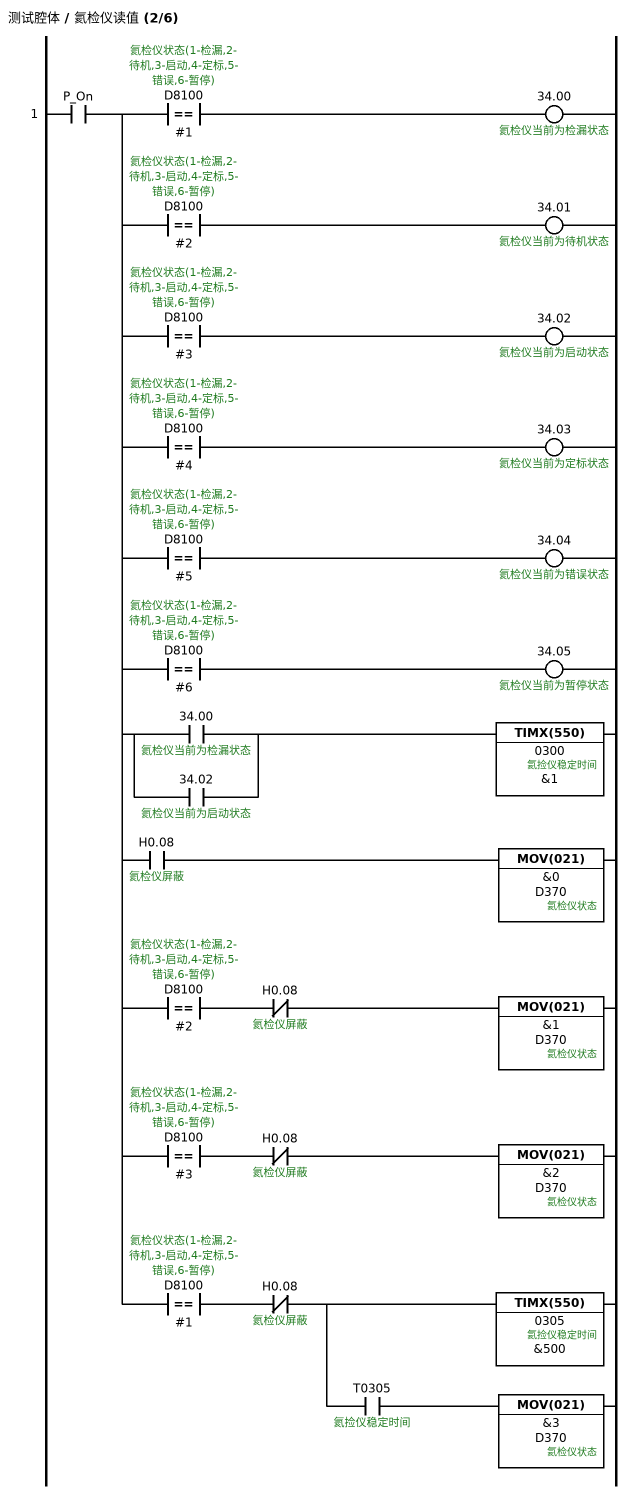
; [picture p144: 测试腔体 / 氦检仪读值, rungs 1-1]
; rung 1
LD P_On
OUT TR0
AND=(300) D8100 #1  ; 氦检仪状态(1-检漏,2-待机,3-启动,4-定标,5-错误,6-暂停)
OUT 34.00  ; 氦检仪当前为检漏状态
LD TR0
AND=(300) D8100 #2  ; 氦检仪状态(1-检漏,2-待机,3-启动,4-定标,5-错误,6-暂停)
OUT 34.01  ; 氦检仪当前为待机状态
LD TR0
AND=(300) D8100 #3  ; 氦检仪状态(1-检漏,2-待机,3-启动,4-定标,5-错误,6-暂停)
OUT 34.02  ; 氦检仪当前为启动状态
LD TR0
AND=(300) D8100 #4  ; 氦检仪状态(1-检漏,2-待机,3-启动,4-定标,5-错误,6-暂停)
OUT 34.03  ; 氦检仪当前为定标状态
LD TR0
AND=(300) D8100 #5  ; 氦检仪状态(1-检漏,2-待机,3-启动,4-定标,5-错误,6-暂停)
OUT 34.04  ; 氦检仪当前为错误状态
LD TR0
AND=(300) D8100 #6  ; 氦检仪状态(1-检漏,2-待机,3-启动,4-定标,5-错误,6-暂停)
OUT 34.05  ; 氦检仪当前为暂停状态
LD TR0
LD 34.00  ; 氦检仪当前为检漏状态
OR 34.02  ; 氦检仪当前为启动状态
ANDLD
TIMX(550) 0300 &1  ; 氦捡仪稳定时间
LD TR0
AND H0.08  ; 氦检仪屏蔽
MOV(021) &0 D370  ; 氦检仪状态
LD TR0
AND=(300) D8100 #2  ; 氦检仪状态(1-检漏,2-待机,3-启动,4-定标,5-错误,6-暂停)
ANDNOT H0.08  ; 氦检仪屏蔽
MOV(021) &1 D370  ; 氦检仪状态
LD TR0
AND=(300) D8100 #3  ; 氦检仪状态(1-检漏,2-待机,3-启动,4-定标,5-错误,6-暂停)
ANDNOT H0.08  ; 氦检仪屏蔽
MOV(021) &2 D370  ; 氦检仪状态
LD TR0
AND=(300) D8100 #1  ; 氦检仪状态(1-检漏,2-待机,3-启动,4-定标,5-错误,6-暂停)
ANDNOT H0.08  ; 氦检仪屏蔽
TIMX(550) 0305 &500  ; 氦捡仪稳定时间
AND T0305  ; 氦捡仪稳定时间
MOV(021) &3 D370  ; 氦检仪状态

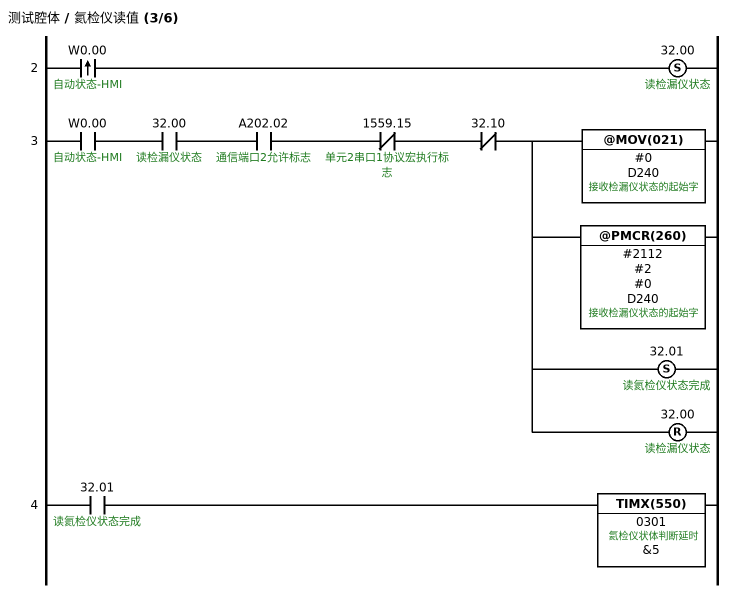
; rung 2
@LD W0.00  ; 自动状态-HMI
SET 32.00  ; 读检漏仪状态
; rung 3
LD W0.00  ; 自动状态-HMI
AND 32.00  ; 读检漏仪状态
AND A202.02  ; 通信端口2允许标志
ANDNOT 1559.15  ; 单元2串口1协议宏执行标志
ANDNOT 32.10
@MOV(021) #0 D240  ; 接收检漏仪状态的起始字
@PMCR(260) #2112 #2 #0 D240  ; 接收检漏仪状态的起始字
SET 32.01  ; 读氦检仪状态完成
RSET 32.00  ; 读检漏仪状态
; rung 4
LD 32.01  ; 读氦检仪状态完成
TIMX(550) 0301 &5  ; 氦检仪状体判断延时

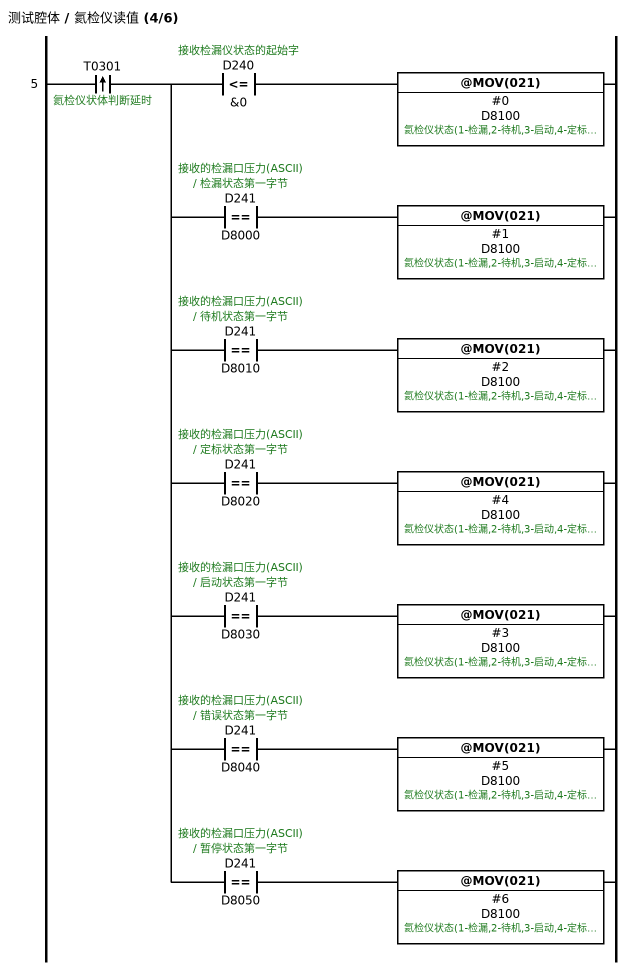
; rung 5
@LD T0301  ; 氦检仪状体判断延时
OUT TR0
AND<=(315) D240 &0  ; 接收检漏仪状态的起始字
@MOV(021) #0 D8100  ; 氦检仪状态(1-检漏,2-待机,3-启动,4-定标,5-错误,6-暂停)
LD TR0
AND=L(301) D241 D8000  ; 接收的检漏口压力(ASCII), 检漏状态第一字节
@MOV(021) #1 D8100  ; 氦检仪状态(1-检漏,2-待机,3-启动,4-定标,5-错误,6-暂停)
LD TR0
AND=L(301) D241 D8010  ; 接收的检漏口压力(ASCII), 待机状态第一字节
@MOV(021) #2 D8100  ; 氦检仪状态(1-检漏,2-待机,3-启动,4-定标,5-错误,6-暂停)
LD TR0
AND=L(301) D241 D8020  ; 接收的检漏口压力(ASCII), 定标状态第一字节
@MOV(021) #4 D8100  ; 氦检仪状态(1-检漏,2-待机,3-启动,4-定标,5-错误,6-暂停)
LD TR0
AND=L(301) D241 D8030  ; 接收的检漏口压力(ASCII), 启动状态第一字节
@MOV(021) #3 D8100  ; 氦检仪状态(1-检漏,2-待机,3-启动,4-定标,5-错误,6-暂停)
LD TR0
AND=L(301) D241 D8040  ; 接收的检漏口压力(ASCII), 错误状态第一字节
@MOV(021) #5 D8100  ; 氦检仪状态(1-检漏,2-待机,3-启动,4-定标,5-错误,6-暂停)
LD TR0
AND=L(301) D241 D8050  ; 接收的检漏口压力(ASCII), 暂停状态第一字节
@MOV(021) #6 D8100  ; 氦检仪状态(1-检漏,2-待机,3-启动,4-定标,5-错误,6-暂停)

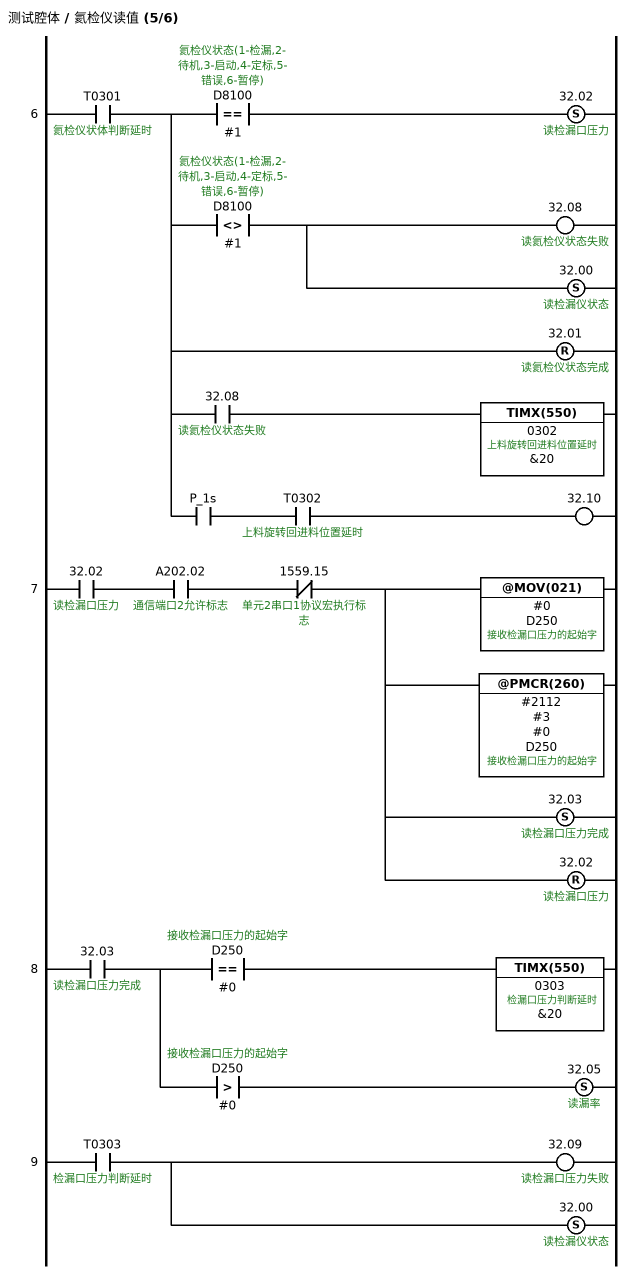
; rung 6
LD T0301  ; 氦检仪状体判断延时
OUT TR0
AND=(300) D8100 #1  ; 氦检仪状态(1-检漏,2-待机,3-启动,4-定标,5-错误,6-暂停)
SET 32.02  ; 读检漏口压力
LD TR0
AND<>(305) D8100 #1  ; 氦检仪状态(1-检漏,2-待机,3-启动,4-定标,5-错误,6-暂停)
OUT 32.08  ; 读氦检仪状态失败
SET 32.00  ; 读检漏仪状态
LD TR0
RSET 32.01  ; 读氦检仪状态完成
AND 32.08  ; 读氦检仪状态失败
TIMX(550) 0302 &20  ; 上料旋转回进料位置延时
LD TR0
AND P_1s
AND T0302  ; 上料旋转回进料位置延时
OUT 32.10
; rung 7
LD 32.02  ; 读检漏口压力
AND A202.02  ; 通信端口2允许标志
ANDNOT 1559.15  ; 单元2串口1协议宏执行标志
@MOV(021) #0 D250  ; 接收检漏口压力的起始字
@PMCR(260) #2112 #3 #0 D250  ; 接收检漏口压力的起始字
SET 32.03  ; 读检漏口压力完成
RSET 32.02  ; 读检漏口压力
; rung 8
LD 32.03  ; 读检漏口压力完成
OUT TR0
AND=(300) D250 #0  ; 接收检漏口压力的起始字
TIMX(550) 0303 &20  ; 检漏口压力判断延时
LD TR0
AND>(320) D250 #0  ; 接收检漏口压力的起始字
SET 32.05  ; 读漏率
; rung 9
LD T0303  ; 检漏口压力判断延时
OUT 32.09  ; 读检漏口压力失败
SET 32.00  ; 读检漏仪状态

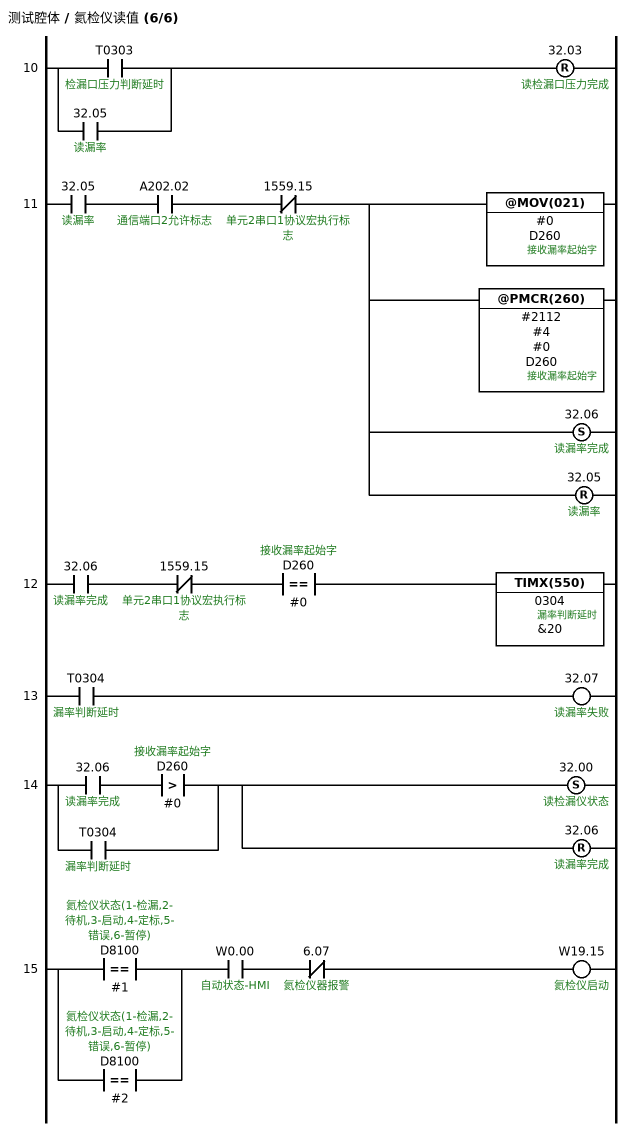
; rung 10
LD T0303  ; 检漏口压力判断延时
OR 32.05  ; 读漏率
RSET 32.03  ; 读检漏口压力完成
; rung 11
LD 32.05  ; 读漏率
AND A202.02  ; 通信端口2允许标志
ANDNOT 1559.15  ; 单元2串口1协议宏执行标志
@MOV(021) #0 D260  ; 接收漏率起始字
@PMCR(260) #2112 #4 #0 D260  ; 接收漏率起始字
SET 32.06  ; 读漏率完成
RSET 32.05  ; 读漏率
; rung 12
LD 32.06  ; 读漏率完成
ANDNOT 1559.15  ; 单元2串口1协议宏执行标志
AND=(300) D260 #0  ; 接收漏率起始字
TIMX(550) 0304 &20  ; 漏率判断延时
; rung 13
LD T0304  ; 漏率判断延时
OUT 32.07  ; 读漏率失败
; rung 14
LD 32.06  ; 读漏率完成
AND>(320) D260 #0  ; 接收漏率起始字
OR T0304  ; 漏率判断延时
SET 32.00  ; 读检漏仪状态
RSET 32.06  ; 读漏率完成
; rung 15
LD=(300) D8100 #1  ; 氦检仪状态(1-检漏,2-待机,3-启动,4-定标,5-错误,6-暂停)
OR=(300) D8100 #2  ; 氦检仪状态(1-检漏,2-待机,3-启动,4-定标,5-错误,6-暂停)
AND W0.00  ; 自动状态-HMI
ANDNOT 6.07  ; 氦检仪器报警
OUT W19.15  ; 氦检仪启动

### Section 外部输出_腔体状态

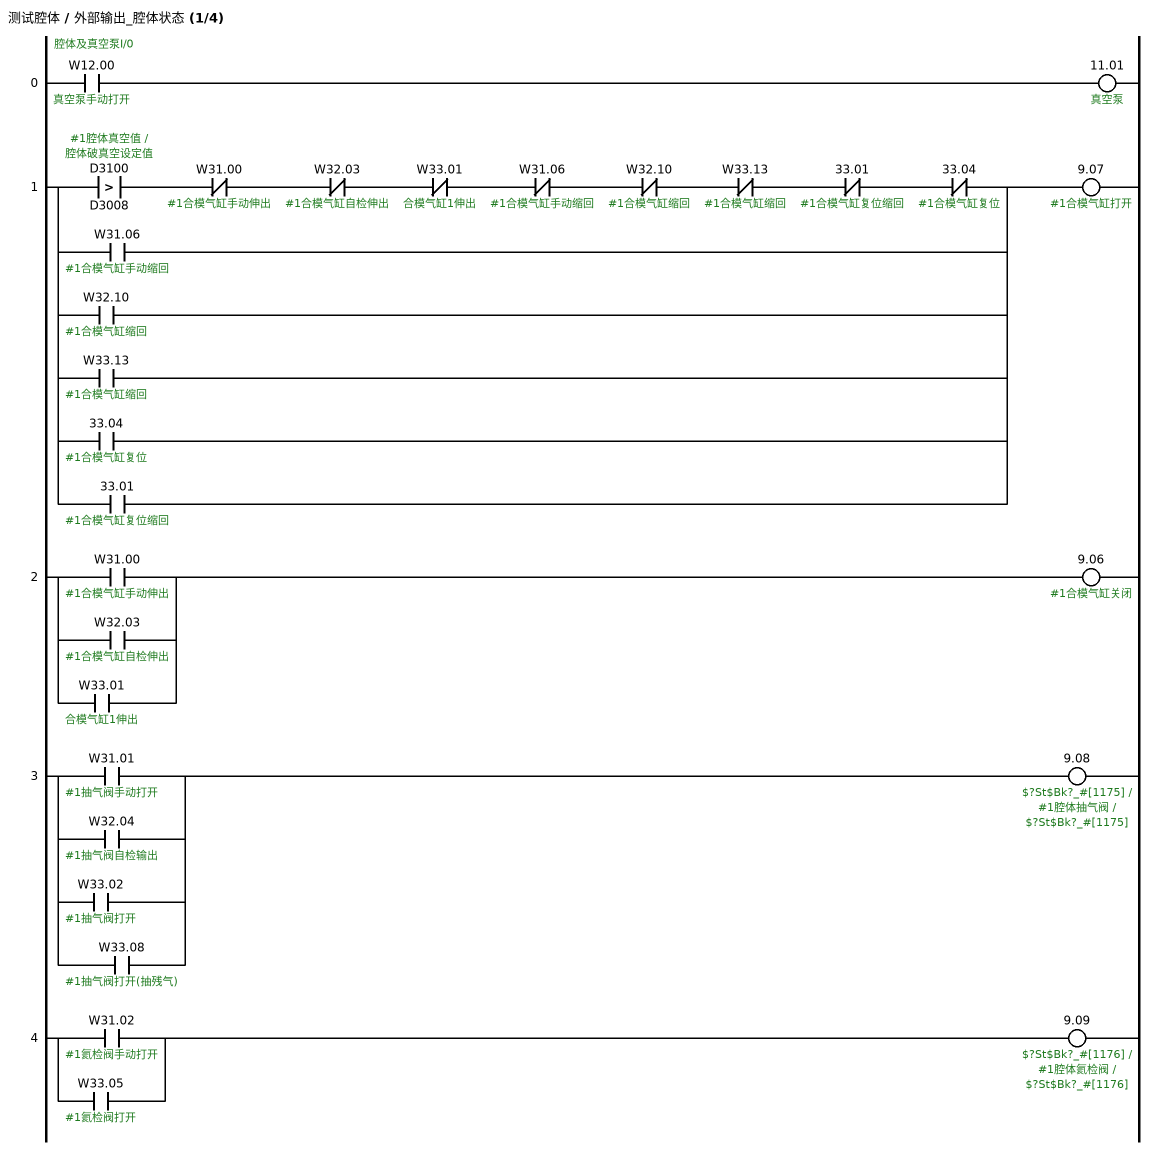
; rung 0: 腔体及真空泵I/0
LD W12.00  ; 真空泵手动打开
OUT 11.01  ; 真空泵
; rung 1
LD>F(333) D3100 D3008  ; #1腔体真空值, 腔体破真空设定值
ANDNOT W31.00  ; #1合模气缸手动伸出
ANDNOT W32.03  ; #1合模气缸自检伸出
ANDNOT W33.01  ; 合模气缸1伸出
ANDNOT W31.06  ; #1合模气缸手动缩回
ANDNOT W32.10  ; #1合模气缸缩回
ANDNOT W33.13  ; #1合模气缸缩回
ANDNOT 33.01  ; #1合模气缸复位缩回
ANDNOT 33.04  ; #1合模气缸复位
OR W31.06  ; #1合模气缸手动缩回
OR W32.10  ; #1合模气缸缩回
OR W33.13  ; #1合模气缸缩回
OR 33.04  ; #1合模气缸复位
OR 33.01  ; #1合模气缸复位缩回
OUT 9.07  ; #1合模气缸打开
; rung 2
LD W31.00  ; #1合模气缸手动伸出
OR W32.03  ; #1合模气缸自检伸出
OR W33.01  ; 合模气缸1伸出
OUT 9.06  ; #1合模气缸关闭
; rung 3
LD W31.01  ; #1抽气阀手动打开
OR W32.04  ; #1抽气阀自检输出
OR W33.02  ; #1抽气阀打开
OR W33.08  ; #1抽气阀打开(抽残气)
OUT 9.08  ; $?St$Bk?_#[1175] / #1腔体抽气阀 / $?St$Bk?_#[1175]
; rung 4
LD W31.02  ; #1氦检阀手动打开
OR W33.05  ; #1氦检阀打开
OUT 9.09  ; $?St$Bk?_#[1176] / #1腔体氦检阀 / $?St$Bk?_#[1176]

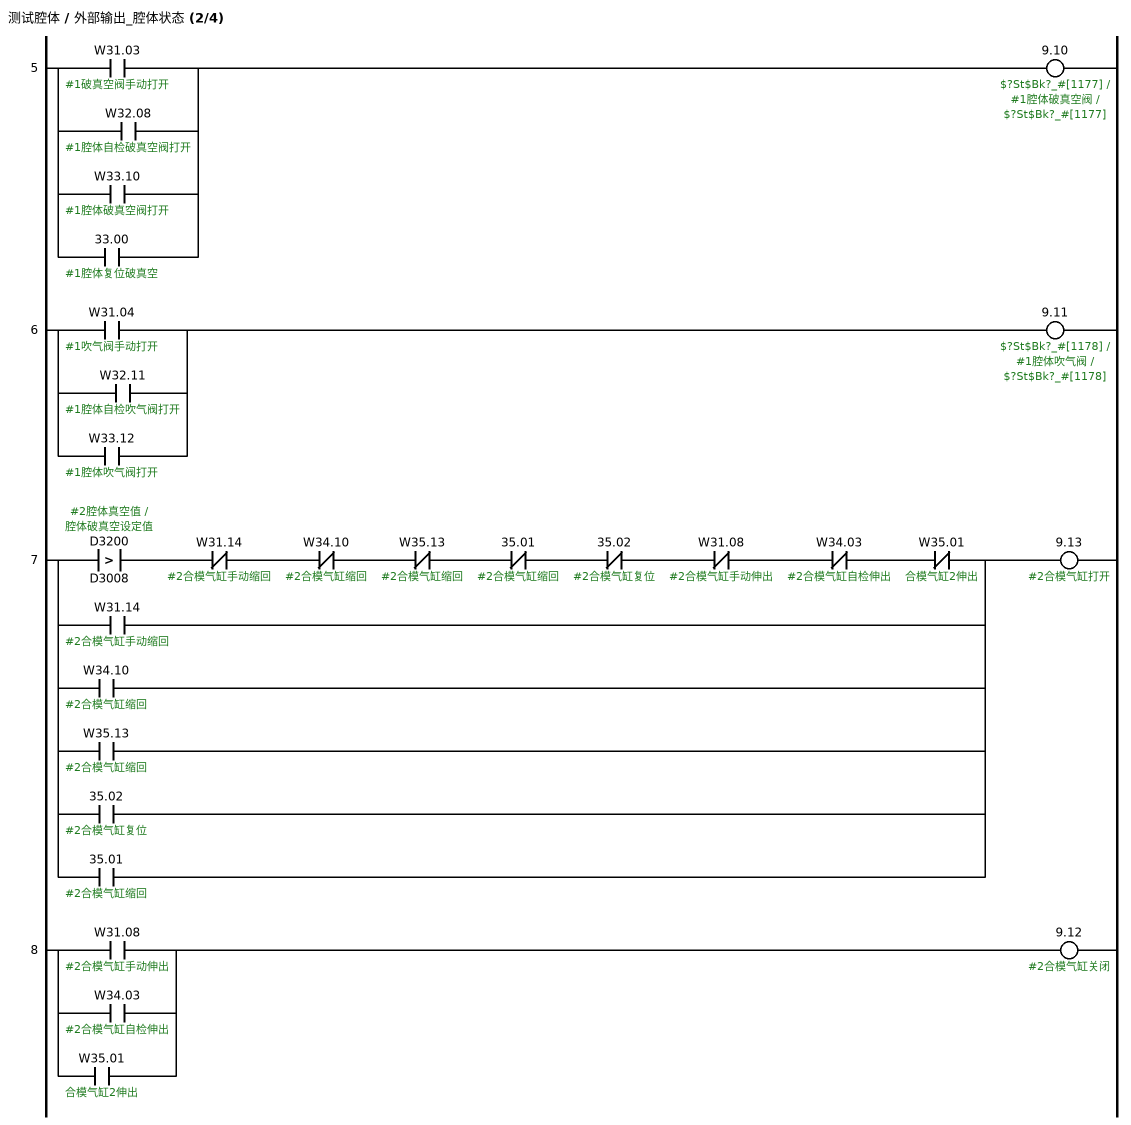
; rung 5
LD W31.03  ; #1破真空阀手动打开
OR W32.08  ; #1腔体自检破真空阀打开
OR W33.10  ; #1腔体破真空阀打开
OR 33.00  ; #1腔体复位破真空
OUT 9.10  ; $?St$Bk?_#[1177] / #1腔体破真空阀 / $?St$Bk?_#[1177]
; rung 6
LD W31.04  ; #1吹气阀手动打开
OR W32.11  ; #1腔体自检吹气阀打开
OR W33.12  ; #1腔体吹气阀打开
OUT 9.11  ; $?St$Bk?_#[1178] / #1腔体吹气阀 / $?St$Bk?_#[1178]
; rung 7
LD>F(333) D3200 D3008  ; #2腔体真空值, 腔体破真空设定值
ANDNOT W31.14  ; #2合模气缸手动缩回
ANDNOT W34.10  ; #2合模气缸缩回
ANDNOT W35.13  ; #2合模气缸缩回
ANDNOT 35.01  ; #2合模气缸缩回
ANDNOT 35.02  ; #2合模气缸复位
ANDNOT W31.08  ; #2合模气缸手动伸出
ANDNOT W34.03  ; #2合模气缸自检伸出
ANDNOT W35.01  ; 合模气缸2伸出
OR W31.14  ; #2合模气缸手动缩回
OR W34.10  ; #2合模气缸缩回
OR W35.13  ; #2合模气缸缩回
OR 35.02  ; #2合模气缸复位
OR 35.01  ; #2合模气缸缩回
OUT 9.13  ; #2合模气缸打开
; rung 8
LD W31.08  ; #2合模气缸手动伸出
OR W34.03  ; #2合模气缸自检伸出
OR W35.01  ; 合模气缸2伸出
OUT 9.12  ; #2合模气缸关闭

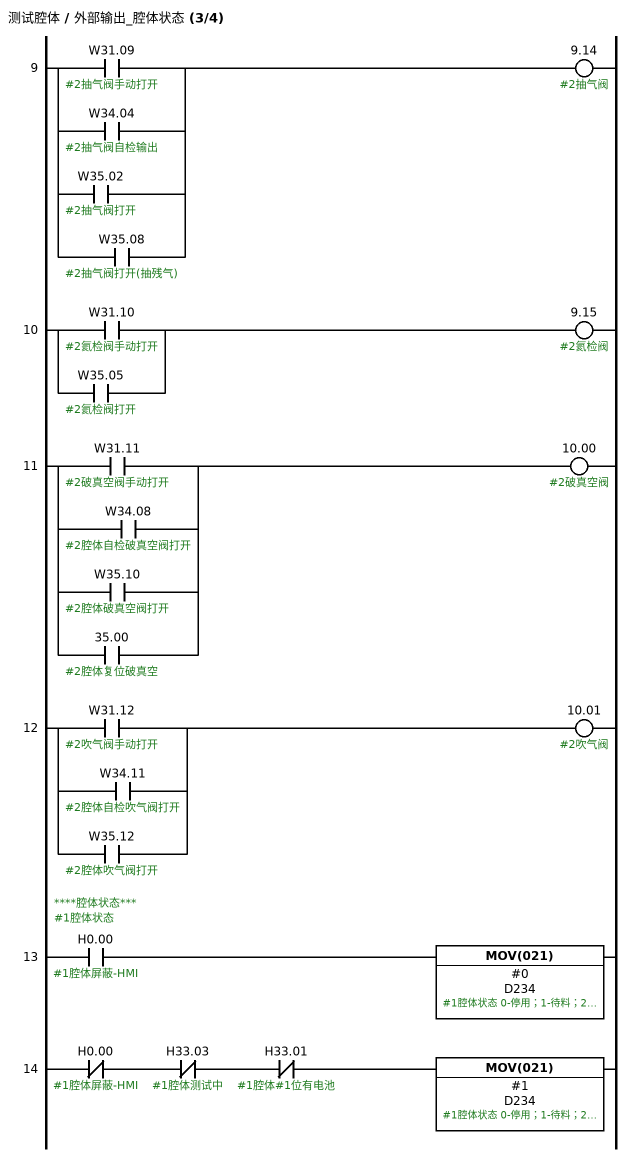
; rung 9
LD W31.09  ; #2抽气阀手动打开
OR W34.04  ; #2抽气阀自检输出
OR W35.02  ; #2抽气阀打开
OR W35.08  ; #2抽气阀打开(抽残气)
OUT 9.14  ; #2抽气阀
; rung 10
LD W31.10  ; #2氦检阀手动打开
OR W35.05  ; #2氦检阀打开
OUT 9.15  ; #2氦检阀
; rung 11
LD W31.11  ; #2破真空阀手动打开
OR W34.08  ; #2腔体自检破真空阀打开
OR W35.10  ; #2腔体破真空阀打开
OR 35.00  ; #2腔体复位破真空
OUT 10.00  ; #2破真空阀
; rung 12
LD W31.12  ; #2吹气阀手动打开
OR W34.11  ; #2腔体自检吹气阀打开
OR W35.12  ; #2腔体吹气阀打开
OUT 10.01  ; #2吹气阀
; rung 13: ****腔体状态*** / #1腔体状态
LD H0.00  ; #1腔体屏蔽-HMI
MOV(021) #0 D234  ; #1腔体状态 0-停用；1-待料；2-测试中；3-测试完成
; rung 14
LDNOT H0.00  ; #1腔体屏蔽-HMI
ANDNOT H33.03  ; #1腔体测试中
ANDNOT H33.01  ; #1腔体#1位有电池
MOV(021) #1 D234  ; #1腔体状态 0-停用；1-待料；2-测试中；3-测试完成

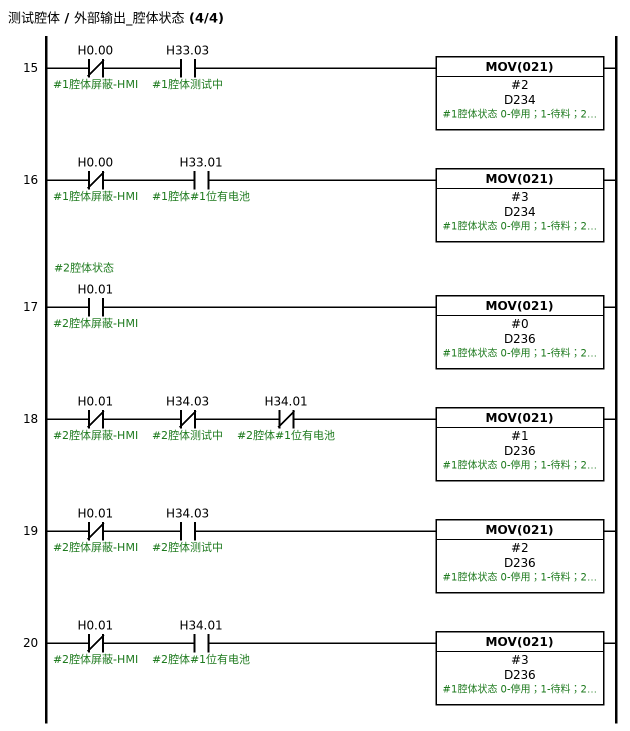
; rung 15
LDNOT H0.00  ; #1腔体屏蔽-HMI
AND H33.03  ; #1腔体测试中
MOV(021) #2 D234  ; #1腔体状态 0-停用；1-待料；2-测试中；3-测试完成
; rung 16
LDNOT H0.00  ; #1腔体屏蔽-HMI
AND H33.01  ; #1腔体#1位有电池
MOV(021) #3 D234  ; #1腔体状态 0-停用；1-待料；2-测试中；3-测试完成
; rung 17: #2腔体状态
LD H0.01  ; #2腔体屏蔽-HMI
MOV(021) #0 D236  ; #1腔体状态 0-停用；1-待料；2-测试中；3-测试完成
; rung 18
LDNOT H0.01  ; #2腔体屏蔽-HMI
ANDNOT H34.03  ; #2腔体测试中
ANDNOT H34.01  ; #2腔体#1位有电池
MOV(021) #1 D236  ; #1腔体状态 0-停用；1-待料；2-测试中；3-测试完成
; rung 19
LDNOT H0.01  ; #2腔体屏蔽-HMI
AND H34.03  ; #2腔体测试中
MOV(021) #2 D236  ; #1腔体状态 0-停用；1-待料；2-测试中；3-测试完成
; rung 20
LDNOT H0.01  ; #2腔体屏蔽-HMI
AND H34.01  ; #2腔体#1位有电池
MOV(021) #3 D236  ; #1腔体状态 0-停用；1-待料；2-测试中；3-测试完成

### Section 报警_复位

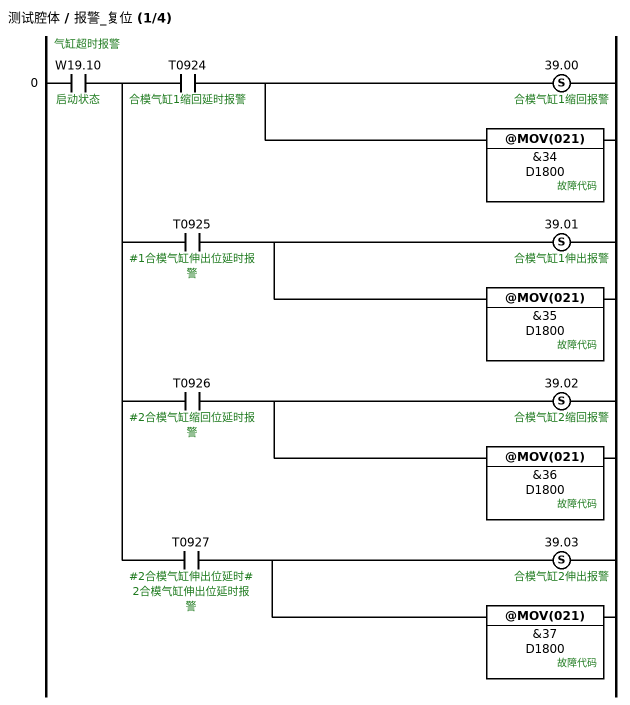
; rung 0: 气缸超时报警
LD W19.10  ; 启动状态
OUT TR0
AND T0924  ; 合模气缸1缩回延时报警
SET 39.00  ; 合模气缸1缩回报警
@MOV(021) &34 D1800  ; 故障代码
LD TR0
AND T0925  ; #1合模气缸伸出位延时报警
SET 39.01  ; 合模气缸1伸出报警
@MOV(021) &35 D1800  ; 故障代码
LD TR0
AND T0926  ; #2合模气缸缩回位延时报警
SET 39.02  ; 合模气缸2缩回报警
@MOV(021) &36 D1800  ; 故障代码
LD TR0
AND T0927  ; #2合模气缸伸出位延时#2合模气缸伸出位延时报警
SET 39.03  ; 合模气缸2伸出报警
@MOV(021) &37 D1800  ; 故障代码

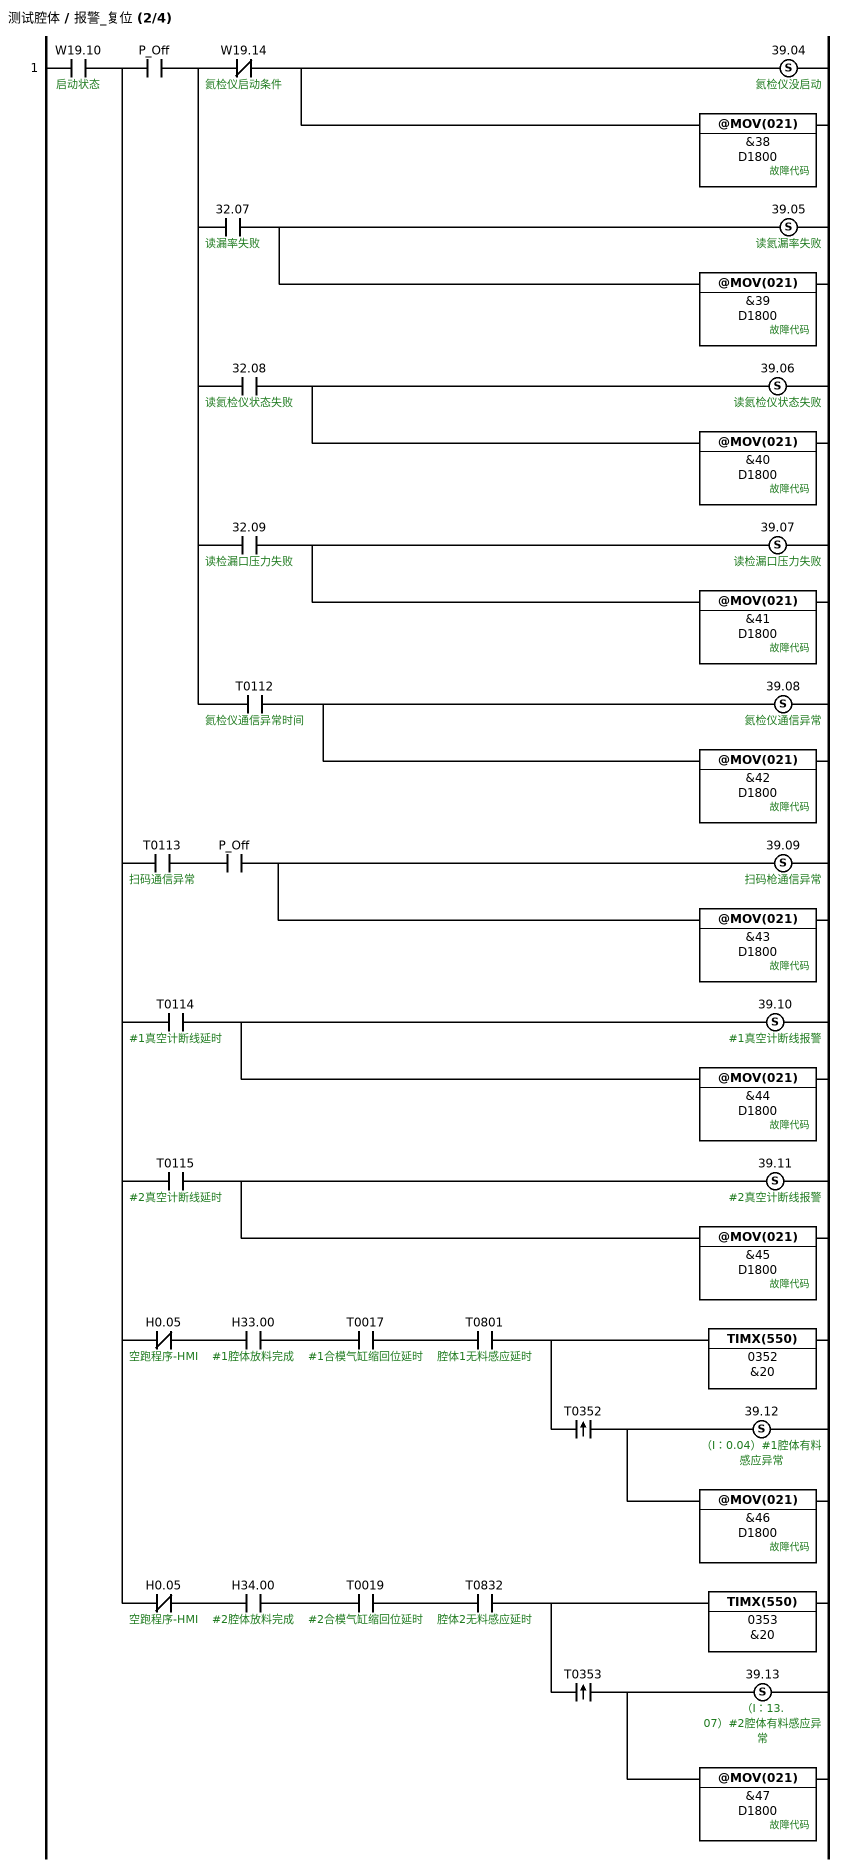
; rung 1
LD W19.10  ; 启动状态
OUT TR0
AND P_Off
OUT TR1
ANDNOT W19.14  ; 氦检仪启动条件
SET 39.04  ; 氦检仪没启动
@MOV(021) &38 D1800  ; 故障代码
LD TR1
AND 32.07  ; 读漏率失败
SET 39.05  ; 读氦漏率失败
@MOV(021) &39 D1800  ; 故障代码
LD TR1
AND 32.08  ; 读氦检仪状态失败
SET 39.06  ; 读氦检仪状态失败
@MOV(021) &40 D1800  ; 故障代码
LD TR1
AND 32.09  ; 读检漏口压力失败
SET 39.07  ; 读检漏口压力失败
@MOV(021) &41 D1800  ; 故障代码
LD TR1
AND T0112  ; 氦检仪通信异常时间
SET 39.08  ; 氦检仪通信异常
@MOV(021) &42 D1800  ; 故障代码
LD TR0
AND T0113  ; 扫码通信异常
AND P_Off
SET 39.09  ; 扫码枪通信异常
@MOV(021) &43 D1800  ; 故障代码
LD TR0
AND T0114  ; #1真空计断线延时
SET 39.10  ; #1真空计断线报警
@MOV(021) &44 D1800  ; 故障代码
LD TR0
AND T0115  ; #2真空计断线延时
SET 39.11  ; #2真空计断线报警
@MOV(021) &45 D1800  ; 故障代码
LD TR0
ANDNOT H0.05  ; 空跑程序-HMI
AND H33.00  ; #1腔体放料完成
AND T0017  ; #1合模气缸缩回位延时
AND T0801  ; 腔体1无料感应延时
TIMX(550) 0352 &20
@AND T0352
SET 39.12  ; （I：0.04）#1腔体有料感应异常
@MOV(021) &46 D1800  ; 故障代码
LD TR0
ANDNOT H0.05  ; 空跑程序-HMI
AND H34.00  ; #2腔体放料完成
AND T0019  ; #2合模气缸缩回位延时
AND T0832  ; 腔体2无料感应延时
TIMX(550) 0353 &20
@AND T0353
SET 39.13  ; （I：13.07）#2腔体有料感应异常
@MOV(021) &47 D1800  ; 故障代码

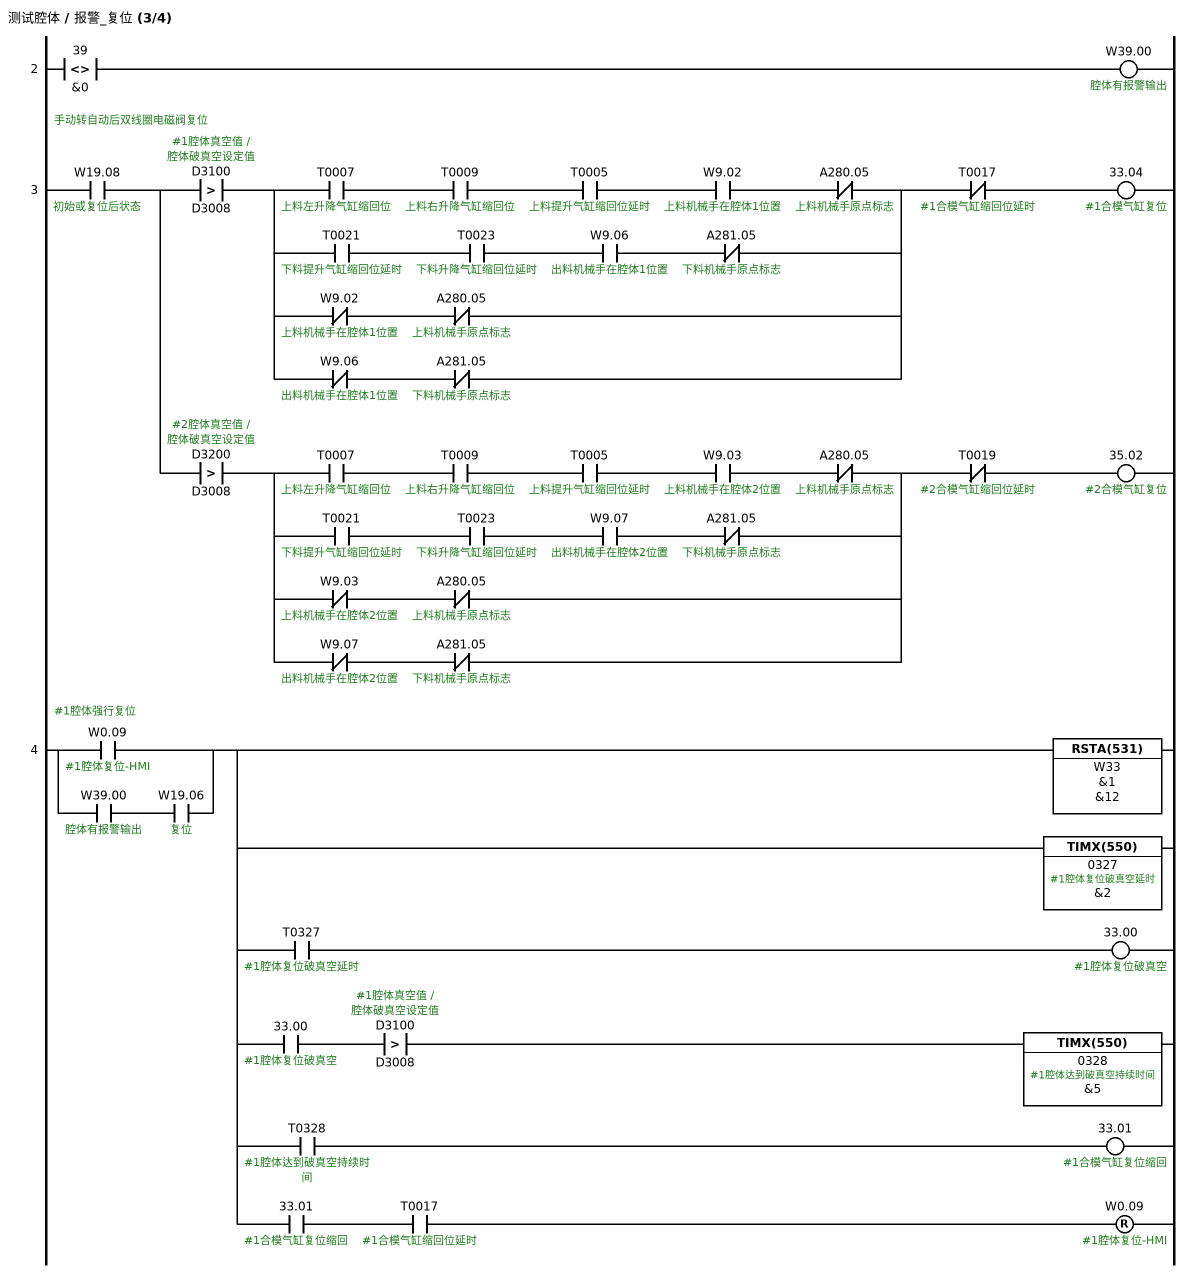
; rung 2
LD<>(305) 39 &0
OUT W39.00  ; 腔体有报警输出
; rung 3: 手动转自动后双线圈电磁阀复位
LD W19.08  ; 初始或复位后状态
OUT TR0
AND>F(333) D3100 D3008  ; #1腔体真空值, 腔体破真空设定值
LD T0007  ; 上料左升降气缸缩回位
AND T0009  ; 上料右升降气缸缩回位
AND T0005  ; 上料提升气缸缩回位延时
AND W9.02  ; 上料机械手在腔体1位置
ANDNOT A280.05  ; 上料机械手原点标志
LD T0021  ; 下料提升气缸缩回位延时
AND T0023  ; 下料升降气缸缩回位延时
AND W9.06  ; 出料机械手在腔体1位置
ANDNOT A281.05  ; 下料机械手原点标志
ORLD
LDNOT W9.02  ; 上料机械手在腔体1位置
ANDNOT A280.05  ; 上料机械手原点标志
ORLD
LDNOT W9.06  ; 出料机械手在腔体1位置
ANDNOT A281.05  ; 下料机械手原点标志
ORLD
ANDLD
ANDNOT T0017  ; #1合模气缸缩回位延时
OUT 33.04  ; #1合模气缸复位
LD TR0
AND>F(333) D3200 D3008  ; #2腔体真空值, 腔体破真空设定值
LD T0007  ; 上料左升降气缸缩回位
AND T0009  ; 上料右升降气缸缩回位
AND T0005  ; 上料提升气缸缩回位延时
AND W9.03  ; 上料机械手在腔体2位置
ANDNOT A280.05  ; 上料机械手原点标志
LD T0021  ; 下料提升气缸缩回位延时
AND T0023  ; 下料升降气缸缩回位延时
AND W9.07  ; 出料机械手在腔体2位置
ANDNOT A281.05  ; 下料机械手原点标志
ORLD
LDNOT W9.03  ; 上料机械手在腔体2位置
ANDNOT A280.05  ; 上料机械手原点标志
ORLD
LDNOT W9.07  ; 出料机械手在腔体2位置
ANDNOT A281.05  ; 下料机械手原点标志
ORLD
ANDLD
ANDNOT T0019  ; #2合模气缸缩回位延时
OUT 35.02  ; #2合模气缸复位
; rung 4: #1腔体强行复位
LD W0.09  ; #1腔体复位-HMI
LD W39.00  ; 腔体有报警输出
AND W19.06  ; 复位
ORLD
OUT TR0
RSTA(531) W33 &1 &12
TIMX(550) 0327 &2  ; #1腔体复位破真空延时
AND T0327  ; #1腔体复位破真空延时
OUT 33.00  ; #1腔体复位破真空
LD TR0
AND 33.00  ; #1腔体复位破真空
AND>F(333) D3100 D3008  ; #1腔体真空值, 腔体破真空设定值
TIMX(550) 0328 &5  ; #1腔体达到破真空持续时间
LD TR0
AND T0328  ; #1腔体达到破真空持续时间
OUT 33.01  ; #1合模气缸复位缩回
LD TR0
AND 33.01  ; #1合模气缸复位缩回
AND T0017  ; #1合模气缸缩回位延时
RSET W0.09  ; #1腔体复位-HMI

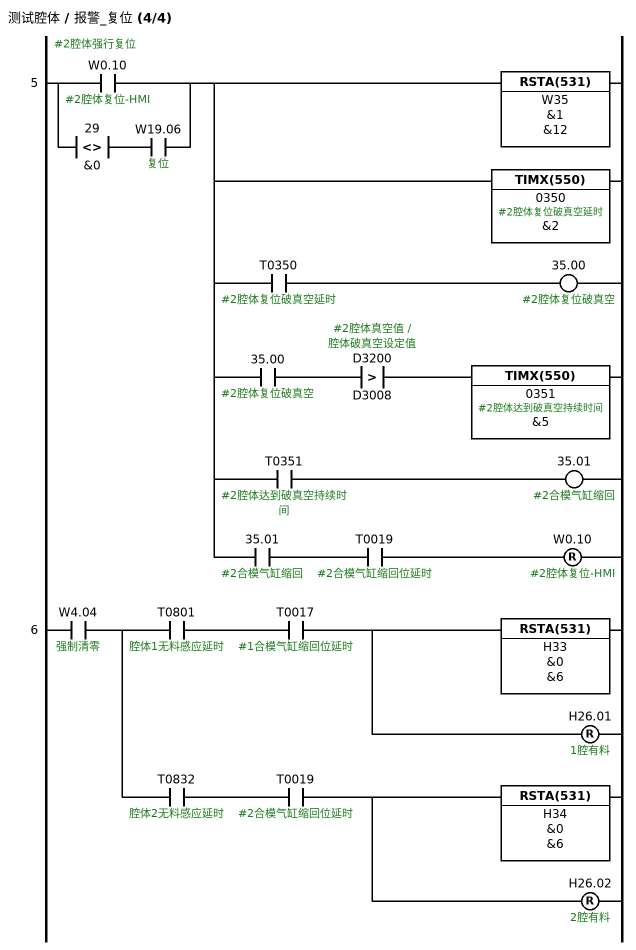
; rung 5: #2腔体强行复位
LD W0.10  ; #2腔体复位-HMI
LD<>(305) 29 &0
AND W19.06  ; 复位
ORLD
OUT TR0
RSTA(531) W35 &1 &12
TIMX(550) 0350 &2  ; #2腔体复位破真空延时
AND T0350  ; #2腔体复位破真空延时
OUT 35.00  ; #2腔体复位破真空
LD TR0
AND 35.00  ; #2腔体复位破真空
AND>F(333) D3200 D3008  ; #2腔体真空值, 腔体破真空设定值
TIMX(550) 0351 &5  ; #2腔体达到破真空持续时间
LD TR0
AND T0351  ; #2腔体达到破真空持续时间
OUT 35.01  ; #2合模气缸缩回
LD TR0
AND 35.01  ; #2合模气缸缩回
AND T0019  ; #2合模气缸缩回位延时
RSET W0.10  ; #2腔体复位-HMI
; rung 6
LD W4.04  ; 强制清零
OUT TR0
AND T0801  ; 腔体1无料感应延时
AND T0017  ; #1合模气缸缩回位延时
RSTA(531) H33 &0 &6
RSET H26.01  ; 1腔有料
LD TR0
AND T0832  ; 腔体2无料感应延时
AND T0019  ; #2合模气缸缩回位延时
RSTA(531) H34 &0 &6
RSET H26.02  ; 2腔有料

### Section END
; rung 0
END(001)

## Program 下料机械手 (cyclic task 4)

### Section 下料机械手手动

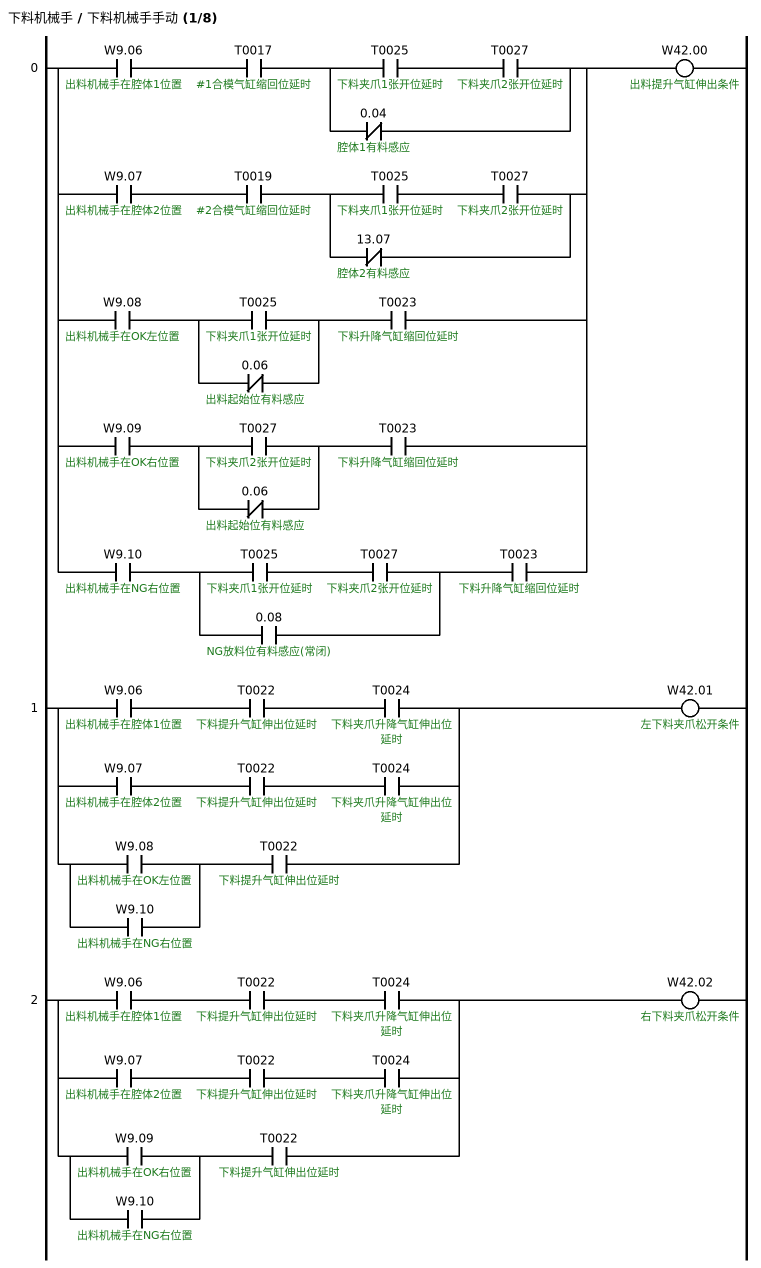
; rung 0
LD W9.06  ; 出料机械手在腔体1位置
AND T0017  ; #1合模气缸缩回位延时
LD T0025  ; 下料夹爪1张开位延时
AND T0027  ; 下料夹爪2张开位延时
ORNOT 0.04  ; 腔体1有料感应
ANDLD
LD W9.07  ; 出料机械手在腔体2位置
AND T0019  ; #2合模气缸缩回位延时
LD T0025  ; 下料夹爪1张开位延时
AND T0027  ; 下料夹爪2张开位延时
ORNOT 13.07  ; 腔体2有料感应
ANDLD
ORLD
LD W9.08  ; 出料机械手在OK左位置
LD T0025  ; 下料夹爪1张开位延时
ORNOT 0.06  ; 出料起始位有料感应
ANDLD
AND T0023  ; 下料升降气缸缩回位延时
ORLD
LD W9.09  ; 出料机械手在OK右位置
LD T0027  ; 下料夹爪2张开位延时
ORNOT 0.06  ; 出料起始位有料感应
ANDLD
AND T0023  ; 下料升降气缸缩回位延时
ORLD
LD W9.10  ; 出料机械手在NG右位置
LD T0025  ; 下料夹爪1张开位延时
AND T0027  ; 下料夹爪2张开位延时
OR 0.08  ; NG放料位有料感应(常闭)
ANDLD
AND T0023  ; 下料升降气缸缩回位延时
ORLD
OUT W42.00  ; 出料提升气缸伸出条件
; rung 1
LD W9.06  ; 出料机械手在腔体1位置
AND T0022  ; 下料提升气缸伸出位延时
AND T0024  ; 下料夹爪升降气缸伸出位延时
LD W9.07  ; 出料机械手在腔体2位置
AND T0022  ; 下料提升气缸伸出位延时
AND T0024  ; 下料夹爪升降气缸伸出位延时
ORLD
LD W9.08  ; 出料机械手在OK左位置
OR W9.10  ; 出料机械手在NG右位置
AND T0022  ; 下料提升气缸伸出位延时
ORLD
OUT W42.01  ; 左下料夹爪松开条件
; rung 2
LD W9.06  ; 出料机械手在腔体1位置
AND T0022  ; 下料提升气缸伸出位延时
AND T0024  ; 下料夹爪升降气缸伸出位延时
LD W9.07  ; 出料机械手在腔体2位置
AND T0022  ; 下料提升气缸伸出位延时
AND T0024  ; 下料夹爪升降气缸伸出位延时
ORLD
LD W9.09  ; 出料机械手在OK右位置
OR W9.10  ; 出料机械手在NG右位置
AND T0022  ; 下料提升气缸伸出位延时
ORLD
OUT W42.02  ; 右下料夹爪松开条件

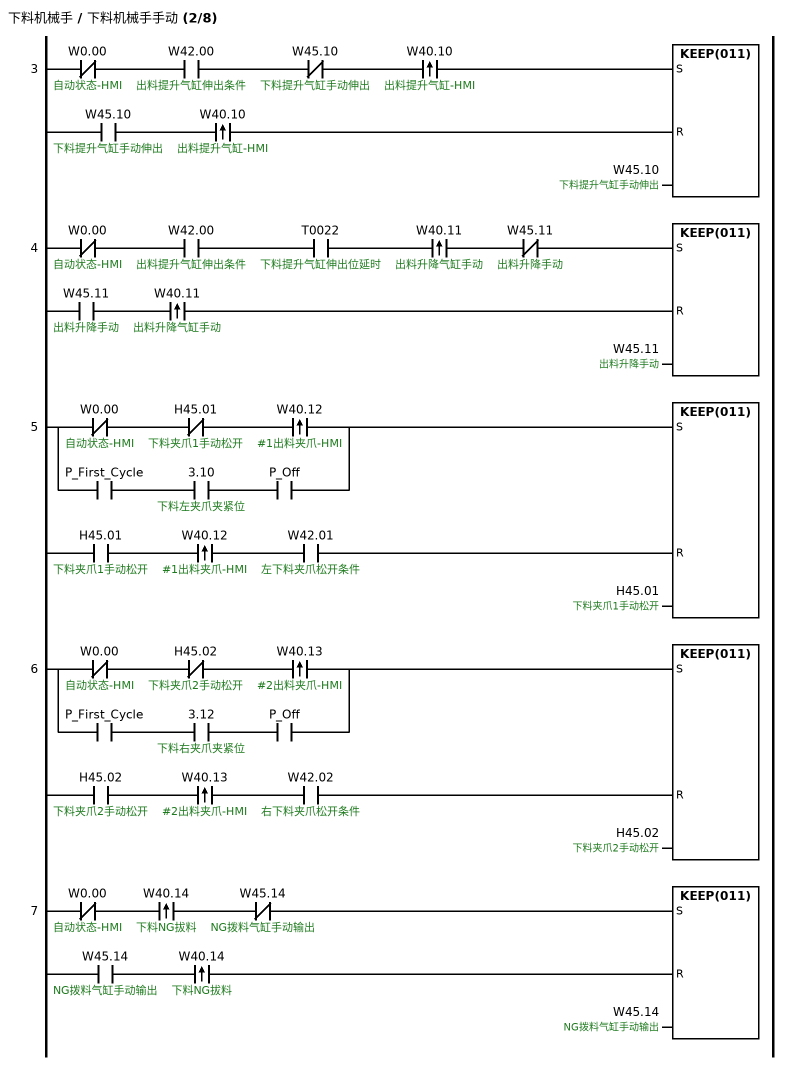
; rung 3
LDNOT W0.00  ; 自动状态-HMI
AND W42.00  ; 出料提升气缸伸出条件
ANDNOT W45.10  ; 下料提升气缸手动伸出
@AND W40.10  ; 出料提升气缸-HMI
LD W45.10  ; 下料提升气缸手动伸出
@AND W40.10  ; 出料提升气缸-HMI
KEEP(011) W45.10  ; 下料提升气缸手动伸出
; rung 4
LDNOT W0.00  ; 自动状态-HMI
AND W42.00  ; 出料提升气缸伸出条件
AND T0022  ; 下料提升气缸伸出位延时
@AND W40.11  ; 出料升降气缸手动
ANDNOT W45.11  ; 出料升降手动
LD W45.11  ; 出料升降手动
@AND W40.11  ; 出料升降气缸手动
KEEP(011) W45.11  ; 出料升降手动
; rung 5
LDNOT W0.00  ; 自动状态-HMI
ANDNOT H45.01  ; 下料夹爪1手动松开
@AND W40.12  ; #1出料夹爪-HMI
LD P_First_Cycle
AND 3.10  ; 下料左夹爪夹紧位
AND P_Off
ORLD
LD H45.01  ; 下料夹爪1手动松开
@AND W40.12  ; #1出料夹爪-HMI
AND W42.01  ; 左下料夹爪松开条件
KEEP(011) H45.01  ; 下料夹爪1手动松开
; rung 6
LDNOT W0.00  ; 自动状态-HMI
ANDNOT H45.02  ; 下料夹爪2手动松开
@AND W40.13  ; #2出料夹爪-HMI
LD P_First_Cycle
AND 3.12  ; 下料右夹爪夹紧位
AND P_Off
ORLD
LD H45.02  ; 下料夹爪2手动松开
@AND W40.13  ; #2出料夹爪-HMI
AND W42.02  ; 右下料夹爪松开条件
KEEP(011) H45.02  ; 下料夹爪2手动松开
; rung 7
LDNOT W0.00  ; 自动状态-HMI
@AND W40.14  ; 下料NG拔料
ANDNOT W45.14  ; NG拨料气缸手动输出
LD W45.14  ; NG拨料气缸手动输出
@AND W40.14  ; 下料NG拔料
KEEP(011) W45.14  ; NG拨料气缸手动输出

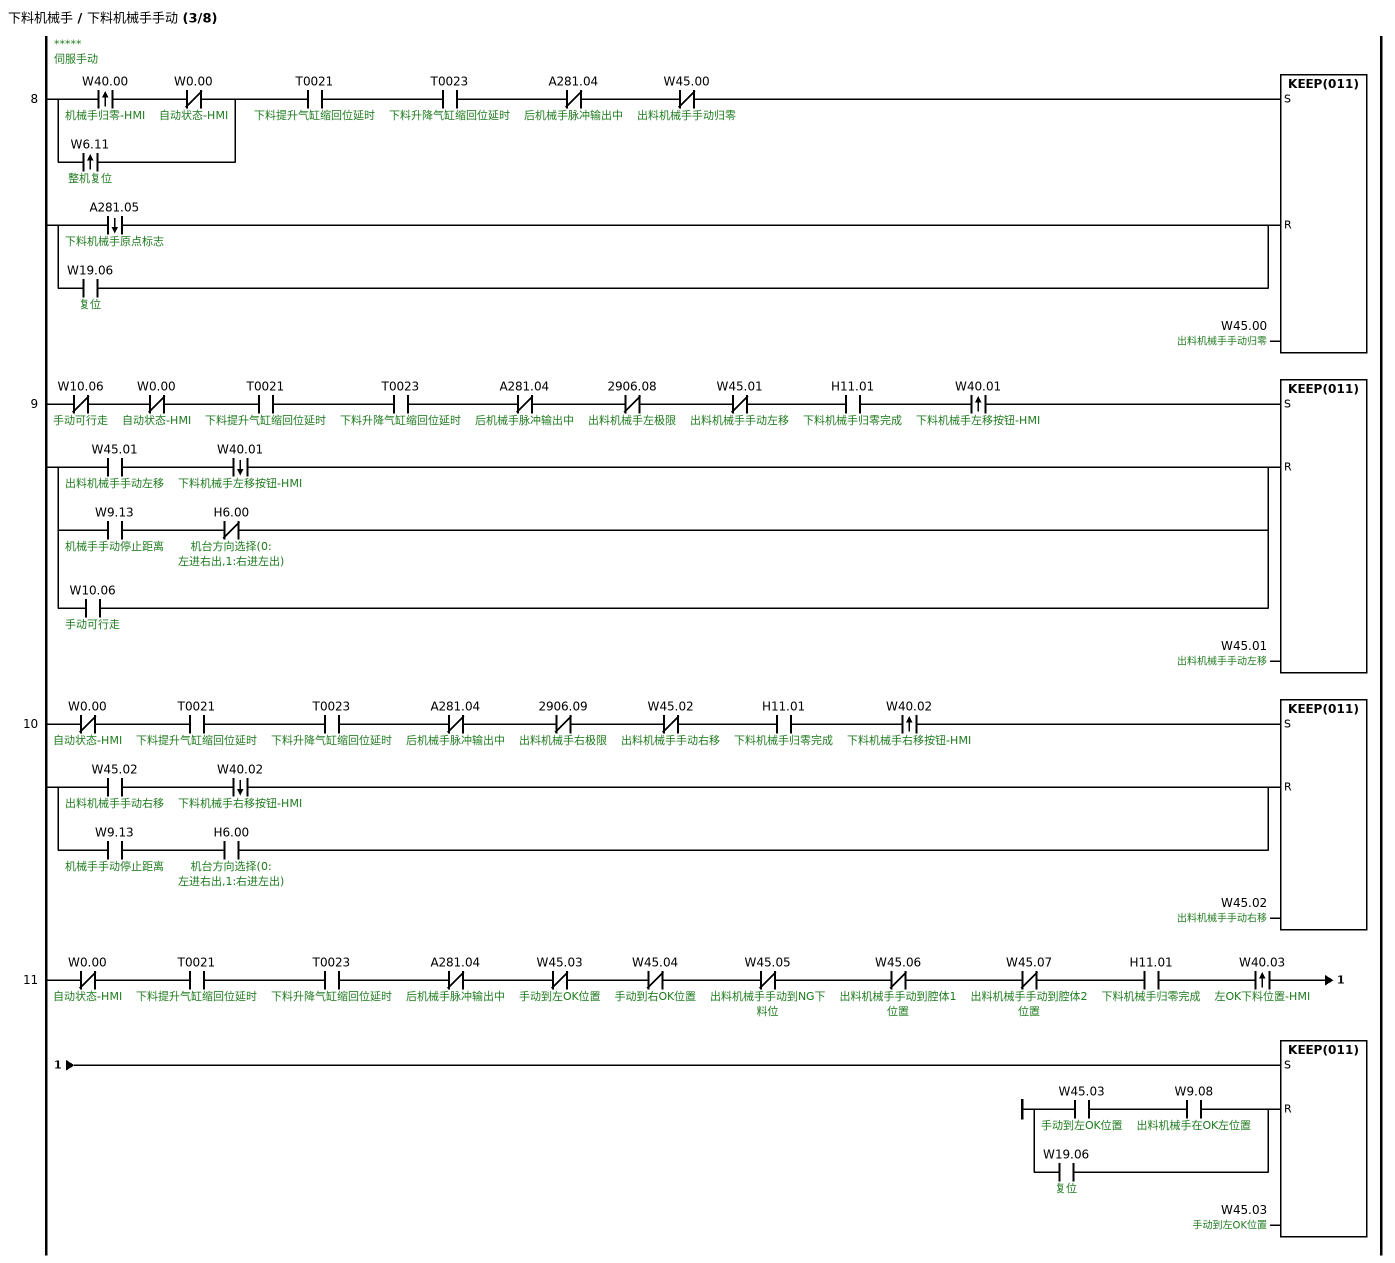
; rung 8: ***** / 伺服手动
@LD W40.00  ; 机械手归零-HMI
ANDNOT W0.00  ; 自动状态-HMI
@OR W6.11  ; 整机复位
AND T0021  ; 下料提升气缸缩回位延时
AND T0023  ; 下料升降气缸缩回位延时
ANDNOT A281.04  ; 后机械手脉冲输出中
ANDNOT W45.00  ; 出料机械手手动归零
%LD A281.05  ; 下料机械手原点标志
OR W19.06  ; 复位
KEEP(011) W45.00  ; 出料机械手手动归零
; rung 9
LDNOT W10.06  ; 手动可行走
ANDNOT W0.00  ; 自动状态-HMI
AND T0021  ; 下料提升气缸缩回位延时
AND T0023  ; 下料升降气缸缩回位延时
ANDNOT A281.04  ; 后机械手脉冲输出中
ANDNOT 2906.08  ; 出料机械手左极限
ANDNOT W45.01  ; 出料机械手手动左移
AND H11.01  ; 下料机械手归零完成
@AND W40.01  ; 下料机械手左移按钮-HMI
LD W45.01  ; 出料机械手手动左移
%AND W40.01  ; 下料机械手左移按钮-HMI
LD W9.13  ; 机械手手动停止距离
ANDNOT H6.00  ; 机台方向选择(0:左进右出,1:右进左出)
ORLD
OR W10.06  ; 手动可行走
KEEP(011) W45.01  ; 出料机械手手动左移
; rung 10
LDNOT W0.00  ; 自动状态-HMI
AND T0021  ; 下料提升气缸缩回位延时
AND T0023  ; 下料升降气缸缩回位延时
ANDNOT A281.04  ; 后机械手脉冲输出中
ANDNOT 2906.09  ; 出料机械手右极限
ANDNOT W45.02  ; 出料机械手手动右移
AND H11.01  ; 下料机械手归零完成
@AND W40.02  ; 下料机械手右移按钮-HMI
LD W45.02  ; 出料机械手手动右移
%AND W40.02  ; 下料机械手右移按钮-HMI
LD W9.13  ; 机械手手动停止距离
AND H6.00  ; 机台方向选择(0:左进右出,1:右进左出)
ORLD
KEEP(011) W45.02  ; 出料机械手手动右移
; rung 11
LDNOT W0.00  ; 自动状态-HMI
AND T0021  ; 下料提升气缸缩回位延时
AND T0023  ; 下料升降气缸缩回位延时
ANDNOT A281.04  ; 后机械手脉冲输出中
ANDNOT W45.03  ; 手动到左OK位置
ANDNOT W45.04  ; 手动到右OK位置
ANDNOT W45.05  ; 出料机械手手动到NG下料位
ANDNOT W45.06  ; 出料机械手手动到腔体1位置
ANDNOT W45.07  ; 出料机械手手动到腔体2位置
AND H11.01  ; 下料机械手归零完成
@AND W40.03  ; 左OK下料位置-HMI
LD W45.03  ; 手动到左OK位置
AND W9.08  ; 出料机械手在OK左位置
OR W19.06  ; 复位
KEEP(011) W45.03  ; 手动到左OK位置

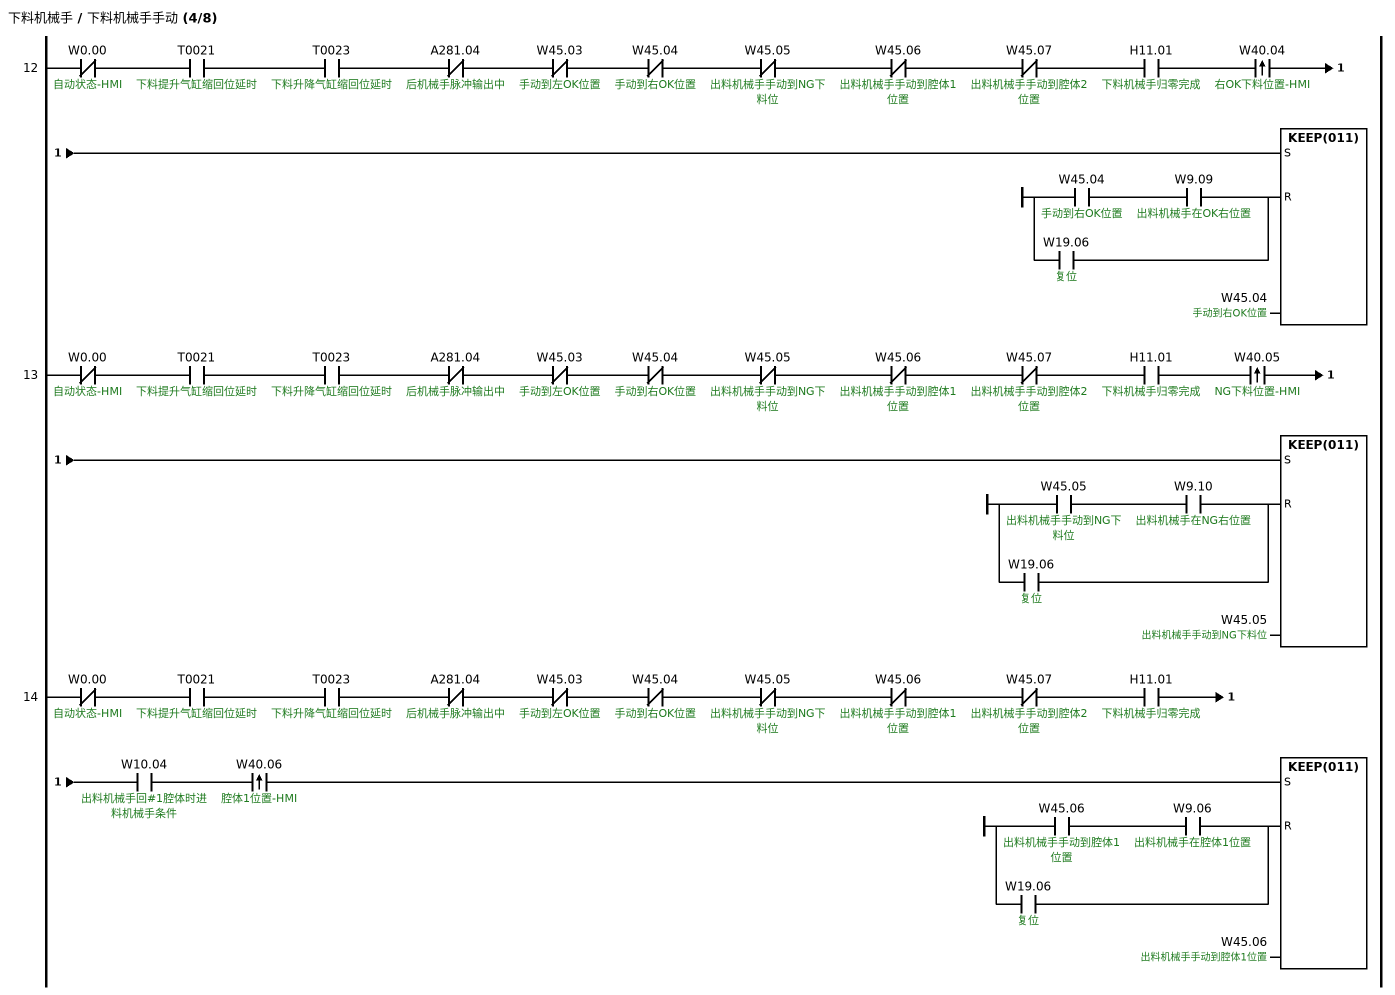
; rung 12
LDNOT W0.00  ; 自动状态-HMI
AND T0021  ; 下料提升气缸缩回位延时
AND T0023  ; 下料升降气缸缩回位延时
ANDNOT A281.04  ; 后机械手脉冲输出中
ANDNOT W45.03  ; 手动到左OK位置
ANDNOT W45.04  ; 手动到右OK位置
ANDNOT W45.05  ; 出料机械手手动到NG下料位
ANDNOT W45.06  ; 出料机械手手动到腔体1位置
ANDNOT W45.07  ; 出料机械手手动到腔体2位置
AND H11.01  ; 下料机械手归零完成
@AND W40.04  ; 右OK下料位置-HMI
LD W45.04  ; 手动到右OK位置
AND W9.09  ; 出料机械手在OK右位置
OR W19.06  ; 复位
KEEP(011) W45.04  ; 手动到右OK位置
; rung 13
LDNOT W0.00  ; 自动状态-HMI
AND T0021  ; 下料提升气缸缩回位延时
AND T0023  ; 下料升降气缸缩回位延时
ANDNOT A281.04  ; 后机械手脉冲输出中
ANDNOT W45.03  ; 手动到左OK位置
ANDNOT W45.04  ; 手动到右OK位置
ANDNOT W45.05  ; 出料机械手手动到NG下料位
ANDNOT W45.06  ; 出料机械手手动到腔体1位置
ANDNOT W45.07  ; 出料机械手手动到腔体2位置
AND H11.01  ; 下料机械手归零完成
@AND W40.05  ; NG下料位置-HMI
LD W45.05  ; 出料机械手手动到NG下料位
AND W9.10  ; 出料机械手在NG右位置
OR W19.06  ; 复位
KEEP(011) W45.05  ; 出料机械手手动到NG下料位
; rung 14
LDNOT W0.00  ; 自动状态-HMI
AND T0021  ; 下料提升气缸缩回位延时
AND T0023  ; 下料升降气缸缩回位延时
ANDNOT A281.04  ; 后机械手脉冲输出中
ANDNOT W45.03  ; 手动到左OK位置
ANDNOT W45.04  ; 手动到右OK位置
ANDNOT W45.05  ; 出料机械手手动到NG下料位
ANDNOT W45.06  ; 出料机械手手动到腔体1位置
ANDNOT W45.07  ; 出料机械手手动到腔体2位置
AND H11.01  ; 下料机械手归零完成
AND W10.04  ; 出料机械手回#1腔体时进料机械手条件
@AND W40.06  ; 腔体1位置-HMI
LD W45.06  ; 出料机械手手动到腔体1位置
AND W9.06  ; 出料机械手在腔体1位置
OR W19.06  ; 复位
KEEP(011) W45.06  ; 出料机械手手动到腔体1位置

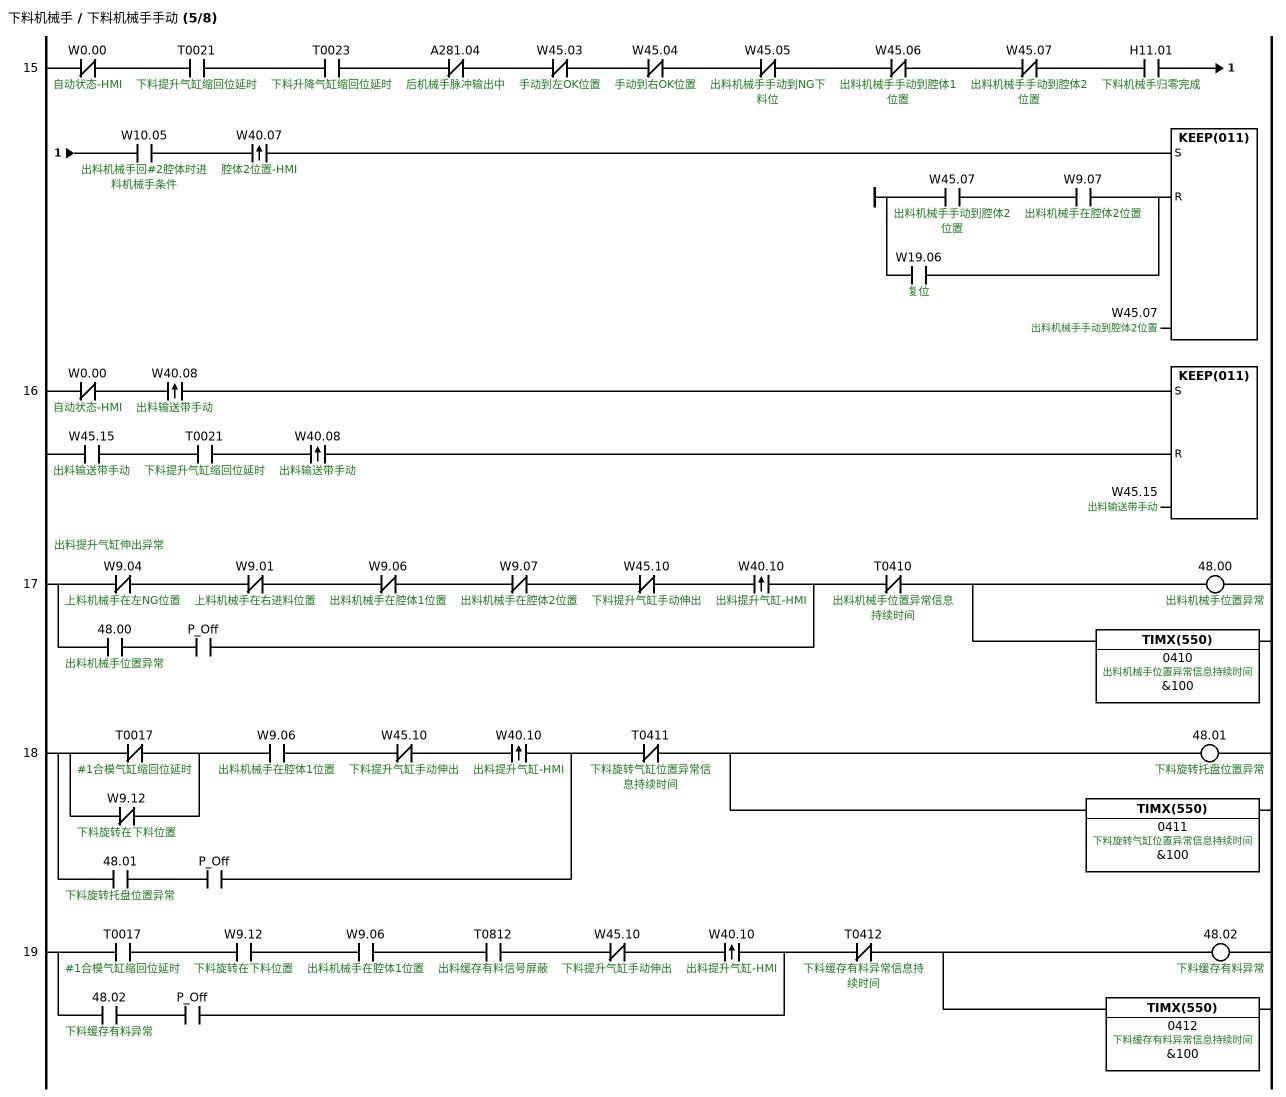
; rung 15
LDNOT W0.00  ; 自动状态-HMI
AND T0021  ; 下料提升气缸缩回位延时
AND T0023  ; 下料升降气缸缩回位延时
ANDNOT A281.04  ; 后机械手脉冲输出中
ANDNOT W45.03  ; 手动到左OK位置
ANDNOT W45.04  ; 手动到右OK位置
ANDNOT W45.05  ; 出料机械手手动到NG下料位
ANDNOT W45.06  ; 出料机械手手动到腔体1位置
ANDNOT W45.07  ; 出料机械手手动到腔体2位置
AND H11.01  ; 下料机械手归零完成
AND W10.05  ; 出料机械手回#2腔体时进料机械手条件
@AND W40.07  ; 腔体2位置-HMI
LD W45.07  ; 出料机械手手动到腔体2位置
AND W9.07  ; 出料机械手在腔体2位置
OR W19.06  ; 复位
KEEP(011) W45.07  ; 出料机械手手动到腔体2位置
; rung 16
LDNOT W0.00  ; 自动状态-HMI
@AND W40.08  ; 出料输送带手动
LD W45.15  ; 出料输送带手动
AND T0021  ; 下料提升气缸缩回位延时
@AND W40.08  ; 出料输送带手动
KEEP(011) W45.15  ; 出料输送带手动
; rung 17: 出料提升气缸伸出异常
LDNOT W9.04  ; 上料机械手在左NG位置
ANDNOT W9.01  ; 上料机械手在右进料位置
ANDNOT W9.06  ; 出料机械手在腔体1位置
ANDNOT W9.07  ; 出料机械手在腔体2位置
ANDNOT W45.10  ; 下料提升气缸手动伸出
@AND W40.10  ; 出料提升气缸-HMI
LD 48.00  ; 出料机械手位置异常
AND P_Off
ORLD
ANDNOT T0410  ; 出料机械手位置异常信息持续时间
OUT 48.00  ; 出料机械手位置异常
TIMX(550) 0410 &100  ; 出料机械手位置异常信息持续时间
; rung 18
LDNOT T0017  ; #1合模气缸缩回位延时
ORNOT W9.12  ; 下料旋转在下料位置
AND W9.06  ; 出料机械手在腔体1位置
ANDNOT W45.10  ; 下料提升气缸手动伸出
@AND W40.10  ; 出料提升气缸-HMI
LD 48.01  ; 下料旋转托盘位置异常
AND P_Off
ORLD
ANDNOT T0411  ; 下料旋转气缸位置异常信息持续时间
OUT 48.01  ; 下料旋转托盘位置异常
TIMX(550) 0411 &100  ; 下料旋转气缸位置异常信息持续时间
; rung 19
LD T0017  ; #1合模气缸缩回位延时
AND W9.12  ; 下料旋转在下料位置
AND W9.06  ; 出料机械手在腔体1位置
AND T0812  ; 出料缓存有料信号屏蔽
ANDNOT W45.10  ; 下料提升气缸手动伸出
@AND W40.10  ; 出料提升气缸-HMI
LD 48.02  ; 下料缓存有料异常
AND P_Off
ORLD
ANDNOT T0412  ; 下料缓存有料异常信息持续时间
OUT 48.02  ; 下料缓存有料异常
TIMX(550) 0412 &100  ; 下料缓存有料异常信息持续时间

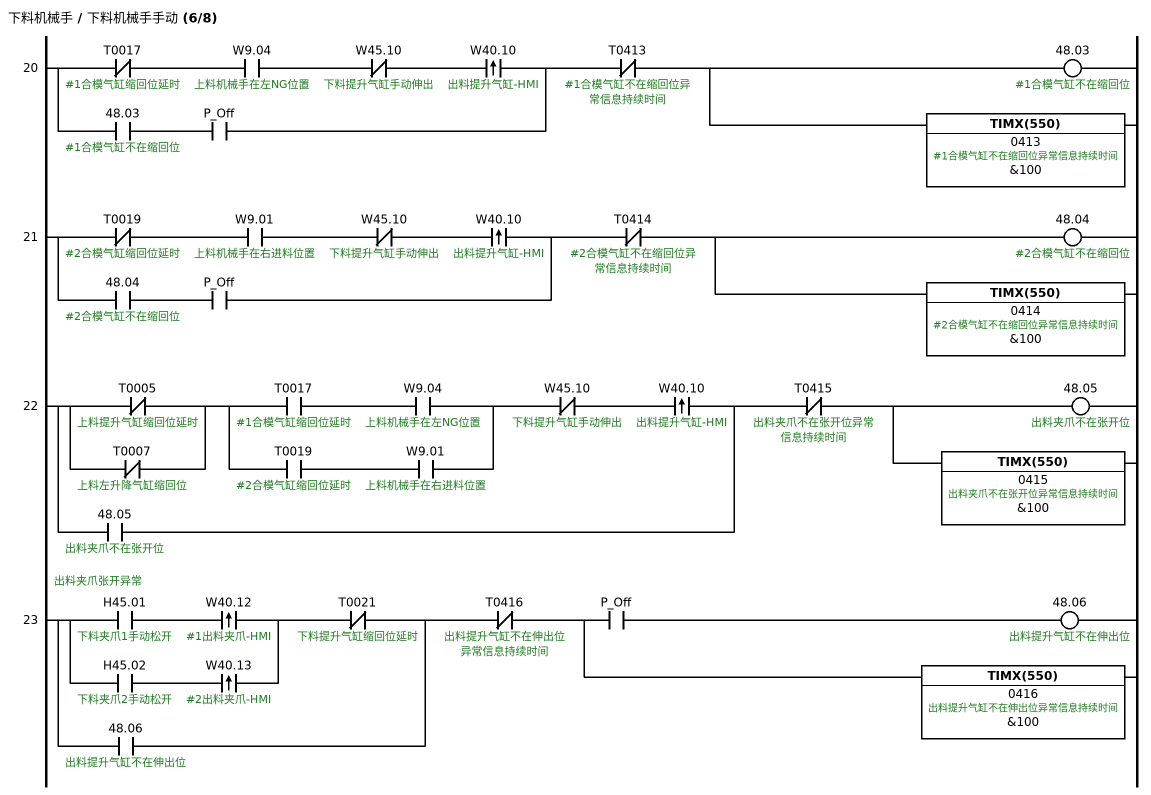
; rung 20
LDNOT T0017  ; #1合模气缸缩回位延时
AND W9.04  ; 上料机械手在左NG位置
ANDNOT W45.10  ; 下料提升气缸手动伸出
@AND W40.10  ; 出料提升气缸-HMI
LD 48.03  ; #1合模气缸不在缩回位
AND P_Off
ORLD
ANDNOT T0413  ; #1合模气缸不在缩回位异常信息持续时间
OUT 48.03  ; #1合模气缸不在缩回位
TIMX(550) 0413 &100  ; #1合模气缸不在缩回位异常信息持续时间
; rung 21
LDNOT T0019  ; #2合模气缸缩回位延时
AND W9.01  ; 上料机械手在右进料位置
ANDNOT W45.10  ; 下料提升气缸手动伸出
@AND W40.10  ; 出料提升气缸-HMI
LD 48.04  ; #2合模气缸不在缩回位
AND P_Off
ORLD
ANDNOT T0414  ; #2合模气缸不在缩回位异常信息持续时间
OUT 48.04  ; #2合模气缸不在缩回位
TIMX(550) 0414 &100  ; #2合模气缸不在缩回位异常信息持续时间
; rung 22
LDNOT T0005  ; 上料提升气缸缩回位延时
ORNOT T0007  ; 上料左升降气缸缩回位
LD T0017  ; #1合模气缸缩回位延时
AND W9.04  ; 上料机械手在左NG位置
LD T0019  ; #2合模气缸缩回位延时
AND W9.01  ; 上料机械手在右进料位置
ORLD
ANDLD
ANDNOT W45.10  ; 下料提升气缸手动伸出
@AND W40.10  ; 出料提升气缸-HMI
OR 48.05  ; 出料夹爪不在张开位
ANDNOT T0415  ; 出料夹爪不在张开位异常信息持续时间
OUT 48.05  ; 出料夹爪不在张开位
TIMX(550) 0415 &100  ; 出料夹爪不在张开位异常信息持续时间
; rung 23: 出料夹爪张开异常
LD H45.01  ; 下料夹爪1手动松开
@AND W40.12  ; #1出料夹爪-HMI
LD H45.02  ; 下料夹爪2手动松开
@AND W40.13  ; #2出料夹爪-HMI
ORLD
ANDNOT T0021  ; 下料提升气缸缩回位延时
OR 48.06  ; 出料提升气缸不在伸出位
ANDNOT T0416  ; 出料提升气缸不在伸出位异常信息持续时间
OUT TR0
AND P_Off
OUT 48.06  ; 出料提升气缸不在伸出位
LD TR0
TIMX(550) 0416 &100  ; 出料提升气缸不在伸出位异常信息持续时间

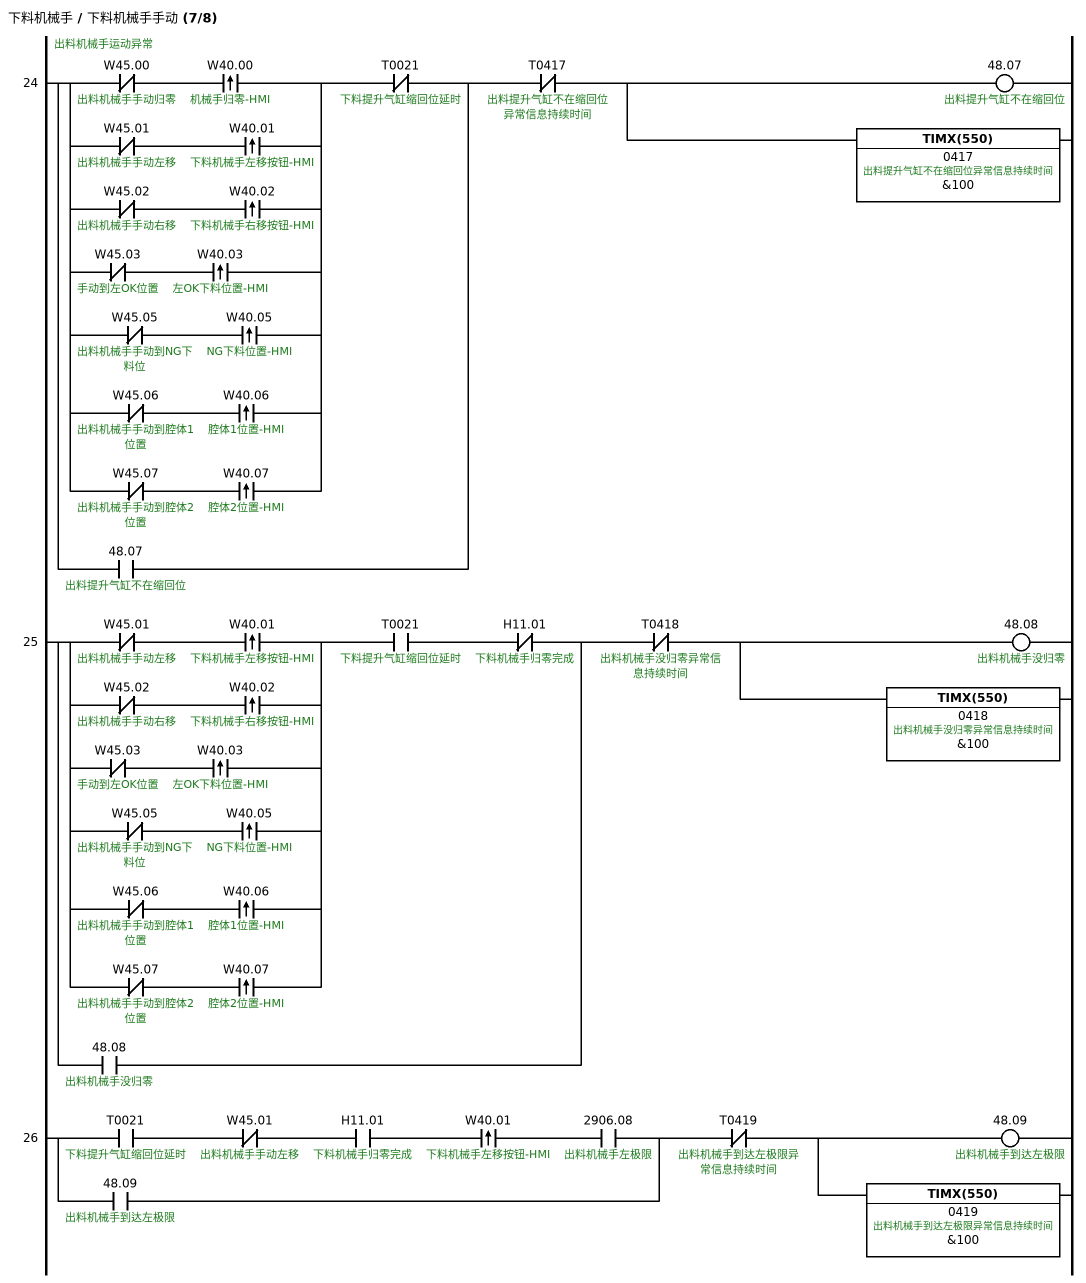
; rung 24: 出料机械手运动异常
LDNOT W45.00  ; 出料机械手手动归零
@AND W40.00  ; 机械手归零-HMI
LDNOT W45.01  ; 出料机械手手动左移
@AND W40.01  ; 下料机械手左移按钮-HMI
ORLD
LDNOT W45.02  ; 出料机械手手动右移
@AND W40.02  ; 下料机械手右移按钮-HMI
ORLD
LDNOT W45.03  ; 手动到左OK位置
@AND W40.03  ; 左OK下料位置-HMI
ORLD
LDNOT W45.05  ; 出料机械手手动到NG下料位
@AND W40.05  ; NG下料位置-HMI
ORLD
LDNOT W45.06  ; 出料机械手手动到腔体1位置
@AND W40.06  ; 腔体1位置-HMI
ORLD
LDNOT W45.07  ; 出料机械手手动到腔体2位置
@AND W40.07  ; 腔体2位置-HMI
ORLD
ANDNOT T0021  ; 下料提升气缸缩回位延时
OR 48.07  ; 出料提升气缸不在缩回位
ANDNOT T0417  ; 出料提升气缸不在缩回位异常信息持续时间
OUT 48.07  ; 出料提升气缸不在缩回位
TIMX(550) 0417 &100  ; 出料提升气缸不在缩回位异常信息持续时间
; rung 25
LDNOT W45.01  ; 出料机械手手动左移
@AND W40.01  ; 下料机械手左移按钮-HMI
LDNOT W45.02  ; 出料机械手手动右移
@AND W40.02  ; 下料机械手右移按钮-HMI
ORLD
LDNOT W45.03  ; 手动到左OK位置
@AND W40.03  ; 左OK下料位置-HMI
ORLD
LDNOT W45.05  ; 出料机械手手动到NG下料位
@AND W40.05  ; NG下料位置-HMI
ORLD
LDNOT W45.06  ; 出料机械手手动到腔体1位置
@AND W40.06  ; 腔体1位置-HMI
ORLD
LDNOT W45.07  ; 出料机械手手动到腔体2位置
@AND W40.07  ; 腔体2位置-HMI
ORLD
AND T0021  ; 下料提升气缸缩回位延时
ANDNOT H11.01  ; 下料机械手归零完成
OR 48.08  ; 出料机械手没归零
ANDNOT T0418  ; 出料机械手没归零异常信息持续时间
OUT 48.08  ; 出料机械手没归零
TIMX(550) 0418 &100  ; 出料机械手没归零异常信息持续时间
; rung 26
LD T0021  ; 下料提升气缸缩回位延时
ANDNOT W45.01  ; 出料机械手手动左移
AND H11.01  ; 下料机械手归零完成
@AND W40.01  ; 下料机械手左移按钮-HMI
AND 2906.08  ; 出料机械手左极限
OR 48.09  ; 出料机械手到达左极限
ANDNOT T0419  ; 出料机械手到达左极限异常信息持续时间
OUT 48.09  ; 出料机械手到达左极限
TIMX(550) 0419 &100  ; 出料机械手到达左极限异常信息持续时间

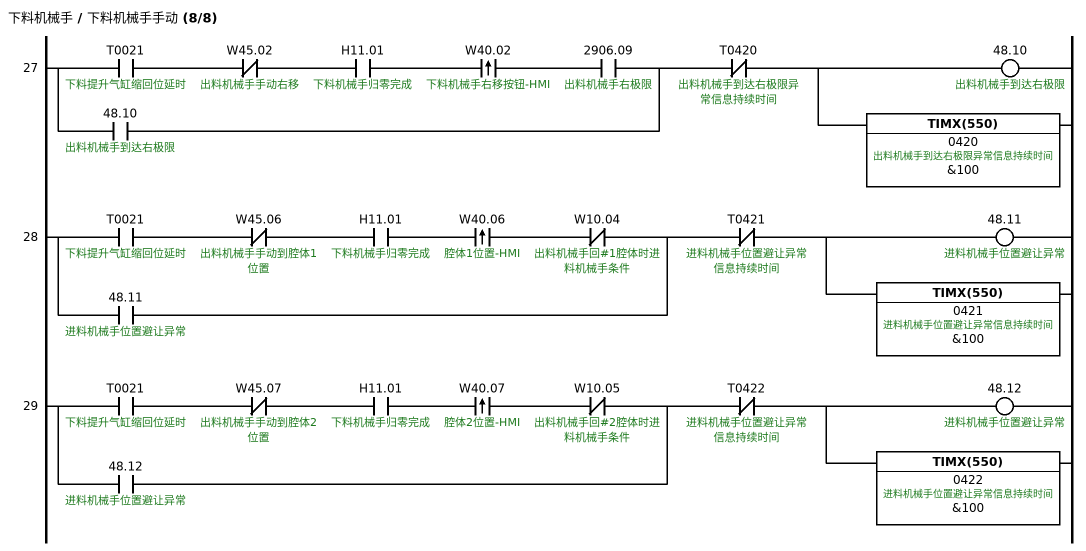
; rung 27
LD T0021  ; 下料提升气缸缩回位延时
ANDNOT W45.02  ; 出料机械手手动右移
AND H11.01  ; 下料机械手归零完成
@AND W40.02  ; 下料机械手右移按钮-HMI
AND 2906.09  ; 出料机械手右极限
OR 48.10  ; 出料机械手到达右极限
ANDNOT T0420  ; 出料机械手到达右极限异常信息持续时间
OUT 48.10  ; 出料机械手到达右极限
TIMX(550) 0420 &100  ; 出料机械手到达右极限异常信息持续时间
; rung 28
LD T0021  ; 下料提升气缸缩回位延时
ANDNOT W45.06  ; 出料机械手手动到腔体1位置
AND H11.01  ; 下料机械手归零完成
@AND W40.06  ; 腔体1位置-HMI
ANDNOT W10.04  ; 出料机械手回#1腔体时进料机械手条件
OR 48.11  ; 进料机械手位置避让异常
ANDNOT T0421  ; 进料机械手位置避让异常信息持续时间
OUT 48.11  ; 进料机械手位置避让异常
TIMX(550) 0421 &100  ; 进料机械手位置避让异常信息持续时间
; rung 29
LD T0021  ; 下料提升气缸缩回位延时
ANDNOT W45.07  ; 出料机械手手动到腔体2位置
AND H11.01  ; 下料机械手归零完成
@AND W40.07  ; 腔体2位置-HMI
ANDNOT W10.05  ; 出料机械手回#2腔体时进料机械手条件
OR 48.12  ; 进料机械手位置避让异常
ANDNOT T0422  ; 进料机械手位置避让异常信息持续时间
OUT 48.12  ; 进料机械手位置避让异常
TIMX(550) 0422 &100  ; 进料机械手位置避让异常信息持续时间

### Section 下料机械手自动

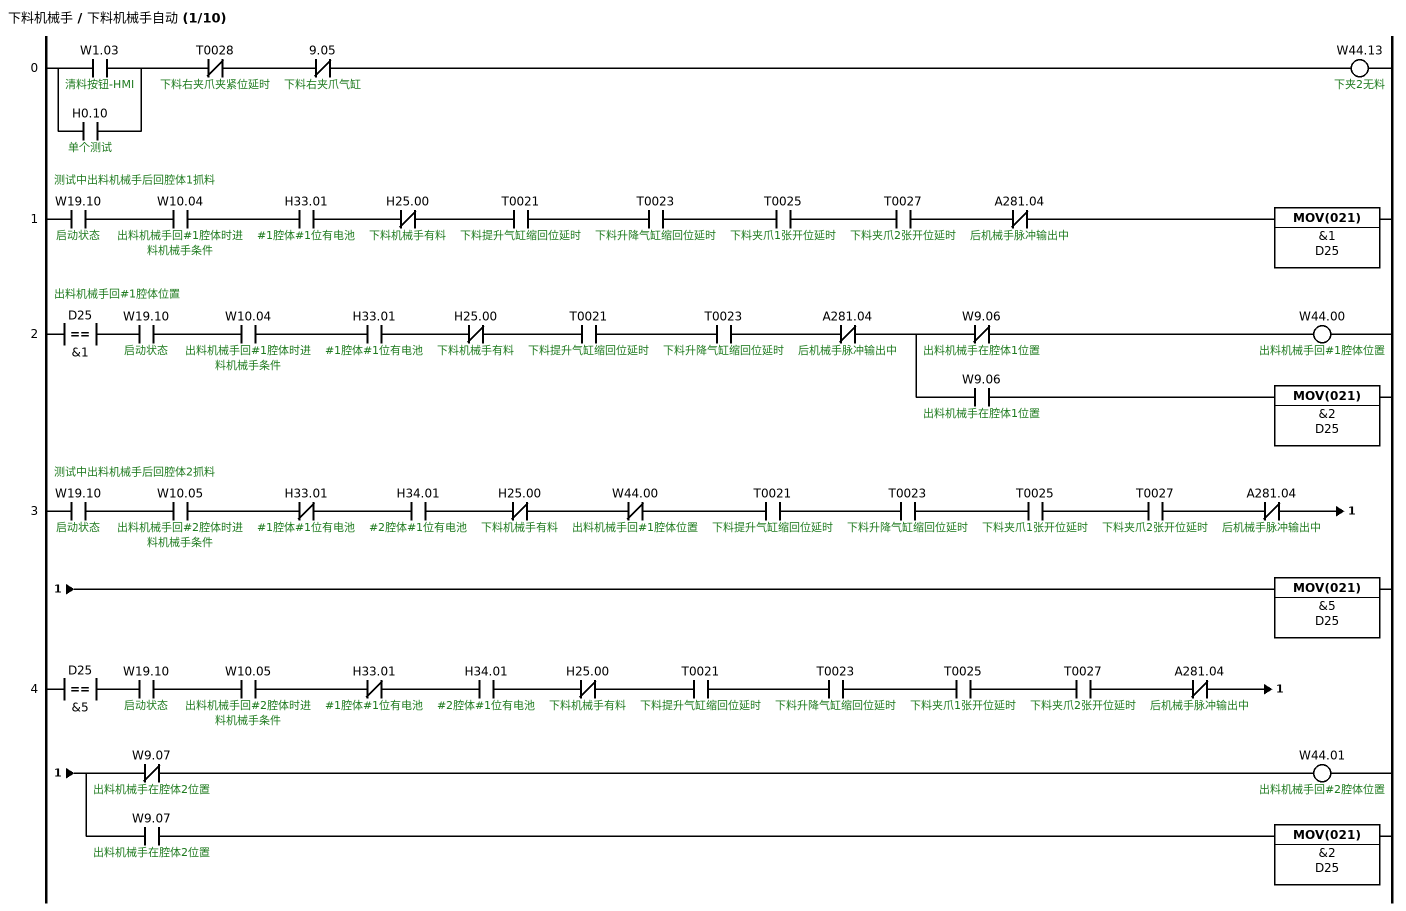
; rung 0
LD W1.03  ; 清料按钮-HMI
OR H0.10  ; 单个测试
ANDNOT T0028  ; 下料右夹爪夹紧位延时
ANDNOT 9.05  ; 下料右夹爪气缸
OUT W44.13  ; 下夹2无料
; rung 1: 测试中出料机械手后回腔体1抓料
LD W19.10  ; 启动状态
AND W10.04  ; 出料机械手回#1腔体时进料机械手条件
AND H33.01  ; #1腔体#1位有电池
ANDNOT H25.00  ; 下料机械手有料
AND T0021  ; 下料提升气缸缩回位延时
AND T0023  ; 下料升降气缸缩回位延时
AND T0025  ; 下料夹爪1张开位延时
AND T0027  ; 下料夹爪2张开位延时
ANDNOT A281.04  ; 后机械手脉冲输出中
MOV(021) &1 D25
; rung 2: 出料机械手回#1腔体位置
LD=(300) D25 &1
AND W19.10  ; 启动状态
AND W10.04  ; 出料机械手回#1腔体时进料机械手条件
AND H33.01  ; #1腔体#1位有电池
ANDNOT H25.00  ; 下料机械手有料
AND T0021  ; 下料提升气缸缩回位延时
AND T0023  ; 下料升降气缸缩回位延时
ANDNOT A281.04  ; 后机械手脉冲输出中
OUT TR0
ANDNOT W9.06  ; 出料机械手在腔体1位置
OUT W44.00  ; 出料机械手回#1腔体位置
LD TR0
AND W9.06  ; 出料机械手在腔体1位置
MOV(021) &2 D25
; rung 3: 测试中出料机械手后回腔体2抓料
LD W19.10  ; 启动状态
AND W10.05  ; 出料机械手回#2腔体时进料机械手条件
ANDNOT H33.01  ; #1腔体#1位有电池
AND H34.01  ; #2腔体#1位有电池
ANDNOT H25.00  ; 下料机械手有料
ANDNOT W44.00  ; 出料机械手回#1腔体位置
AND T0021  ; 下料提升气缸缩回位延时
AND T0023  ; 下料升降气缸缩回位延时
AND T0025  ; 下料夹爪1张开位延时
AND T0027  ; 下料夹爪2张开位延时
ANDNOT A281.04  ; 后机械手脉冲输出中
MOV(021) &5 D25
; rung 4
LD=(300) D25 &5
AND W19.10  ; 启动状态
AND W10.05  ; 出料机械手回#2腔体时进料机械手条件
ANDNOT H33.01  ; #1腔体#1位有电池
AND H34.01  ; #2腔体#1位有电池
ANDNOT H25.00  ; 下料机械手有料
AND T0021  ; 下料提升气缸缩回位延时
AND T0023  ; 下料升降气缸缩回位延时
AND T0025  ; 下料夹爪1张开位延时
AND T0027  ; 下料夹爪2张开位延时
ANDNOT A281.04  ; 后机械手脉冲输出中
OUT TR0
ANDNOT W9.07  ; 出料机械手在腔体2位置
OUT W44.01  ; 出料机械手回#2腔体位置
LD TR0
AND W9.07  ; 出料机械手在腔体2位置
MOV(021) &2 D25

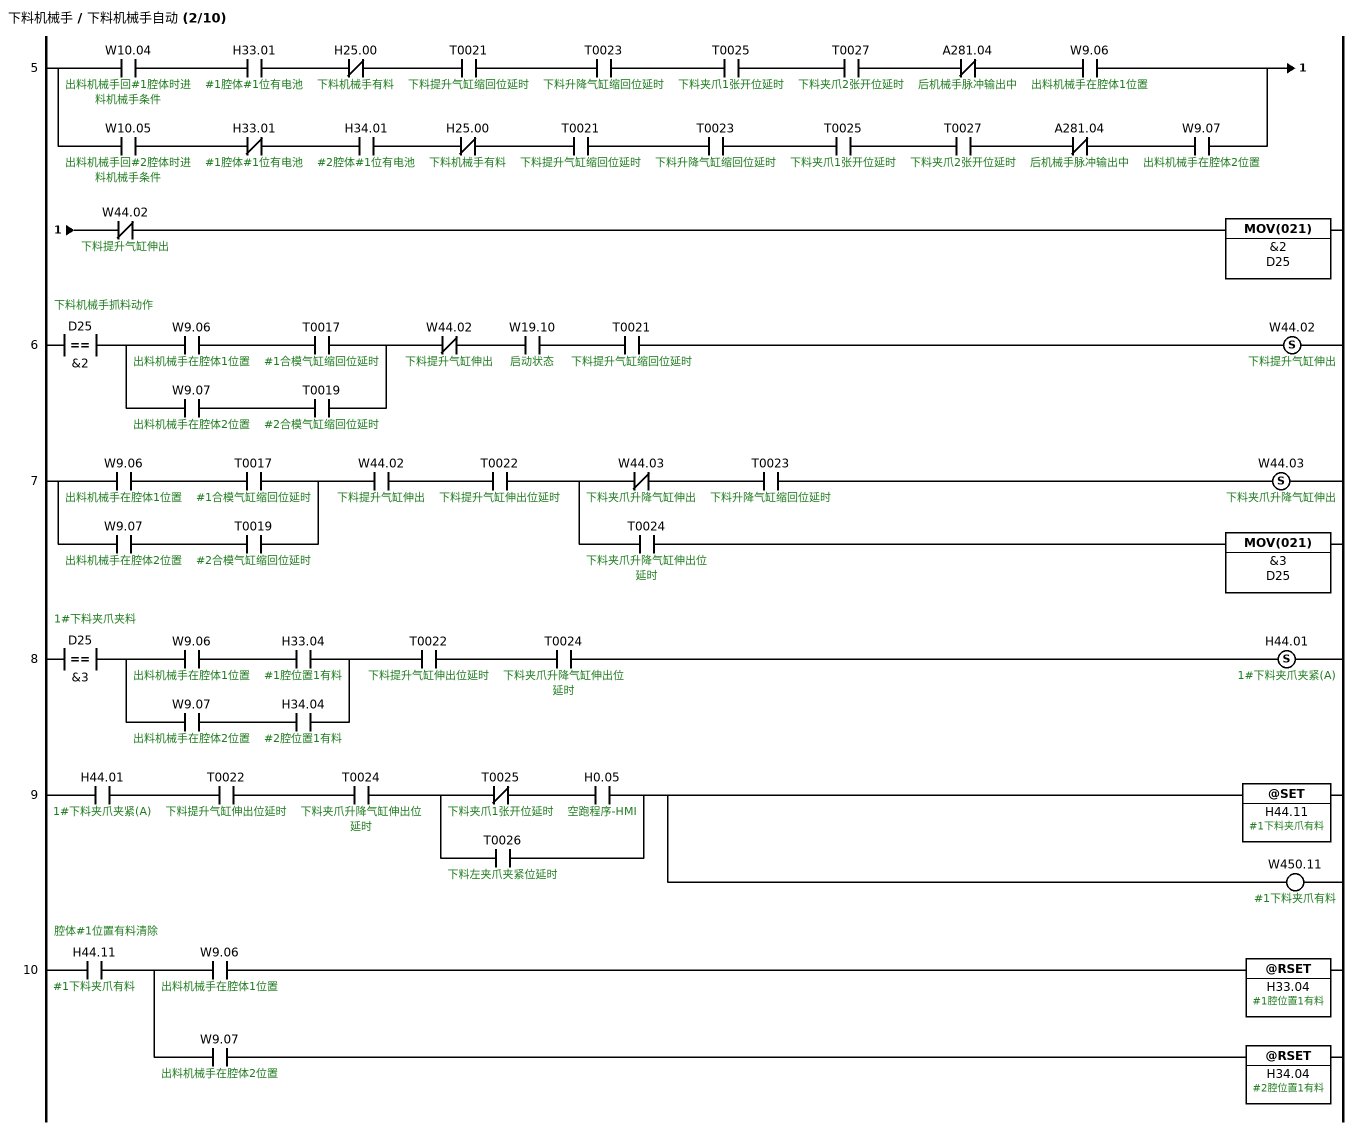
; rung 5
LD W10.04  ; 出料机械手回#1腔体时进料机械手条件
AND H33.01  ; #1腔体#1位有电池
ANDNOT H25.00  ; 下料机械手有料
AND T0021  ; 下料提升气缸缩回位延时
AND T0023  ; 下料升降气缸缩回位延时
AND T0025  ; 下料夹爪1张开位延时
AND T0027  ; 下料夹爪2张开位延时
ANDNOT A281.04  ; 后机械手脉冲输出中
AND W9.06  ; 出料机械手在腔体1位置
LD W10.05  ; 出料机械手回#2腔体时进料机械手条件
ANDNOT H33.01  ; #1腔体#1位有电池
AND H34.01  ; #2腔体#1位有电池
ANDNOT H25.00  ; 下料机械手有料
AND T0021  ; 下料提升气缸缩回位延时
AND T0023  ; 下料升降气缸缩回位延时
AND T0025  ; 下料夹爪1张开位延时
AND T0027  ; 下料夹爪2张开位延时
ANDNOT A281.04  ; 后机械手脉冲输出中
AND W9.07  ; 出料机械手在腔体2位置
ORLD
ANDNOT W44.02  ; 下料提升气缸伸出
MOV(021) &2 D25
; rung 6: 下料机械手抓料动作
LD=(300) D25 &2
LD W9.06  ; 出料机械手在腔体1位置
AND T0017  ; #1合模气缸缩回位延时
LD W9.07  ; 出料机械手在腔体2位置
AND T0019  ; #2合模气缸缩回位延时
ORLD
ANDLD
ANDNOT W44.02  ; 下料提升气缸伸出
AND W19.10  ; 启动状态
AND T0021  ; 下料提升气缸缩回位延时
SET W44.02  ; 下料提升气缸伸出
; rung 7
LD W9.06  ; 出料机械手在腔体1位置
AND T0017  ; #1合模气缸缩回位延时
LD W9.07  ; 出料机械手在腔体2位置
AND T0019  ; #2合模气缸缩回位延时
ORLD
AND W44.02  ; 下料提升气缸伸出
AND T0022  ; 下料提升气缸伸出位延时
OUT TR0
ANDNOT W44.03  ; 下料夹爪升降气缸伸出
AND T0023  ; 下料升降气缸缩回位延时
SET W44.03  ; 下料夹爪升降气缸伸出
LD TR0
AND T0024  ; 下料夹爪升降气缸伸出位延时
MOV(021) &3 D25
; rung 8: 1#下料夹爪夹料
LD=(300) D25 &3
LD W9.06  ; 出料机械手在腔体1位置
AND H33.04  ; #1腔位置1有料
LD W9.07  ; 出料机械手在腔体2位置
AND H34.04  ; #2腔位置1有料
ORLD
ANDLD
AND T0022  ; 下料提升气缸伸出位延时
AND T0024  ; 下料夹爪升降气缸伸出位延时
SET H44.01  ; 1#下料夹爪夹紧(A)
; rung 9
LD H44.01  ; 1#下料夹爪夹紧(A)
AND T0022  ; 下料提升气缸伸出位延时
AND T0024  ; 下料夹爪升降气缸伸出位延时
LDNOT T0025  ; 下料夹爪1张开位延时
AND H0.05  ; 空跑程序-HMI
OR T0026  ; 下料左夹爪夹紧位延时
ANDLD
@SET H44.11  ; #1下料夹爪有料
OUT W450.11  ; #1下料夹爪有料
; rung 10: 腔体#1位置有料清除
LD H44.11  ; #1下料夹爪有料
OUT TR0
AND W9.06  ; 出料机械手在腔体1位置
@RSET H33.04  ; #1腔位置1有料
LD TR0
AND W9.07  ; 出料机械手在腔体2位置
@RSET H34.04  ; #2腔位置1有料

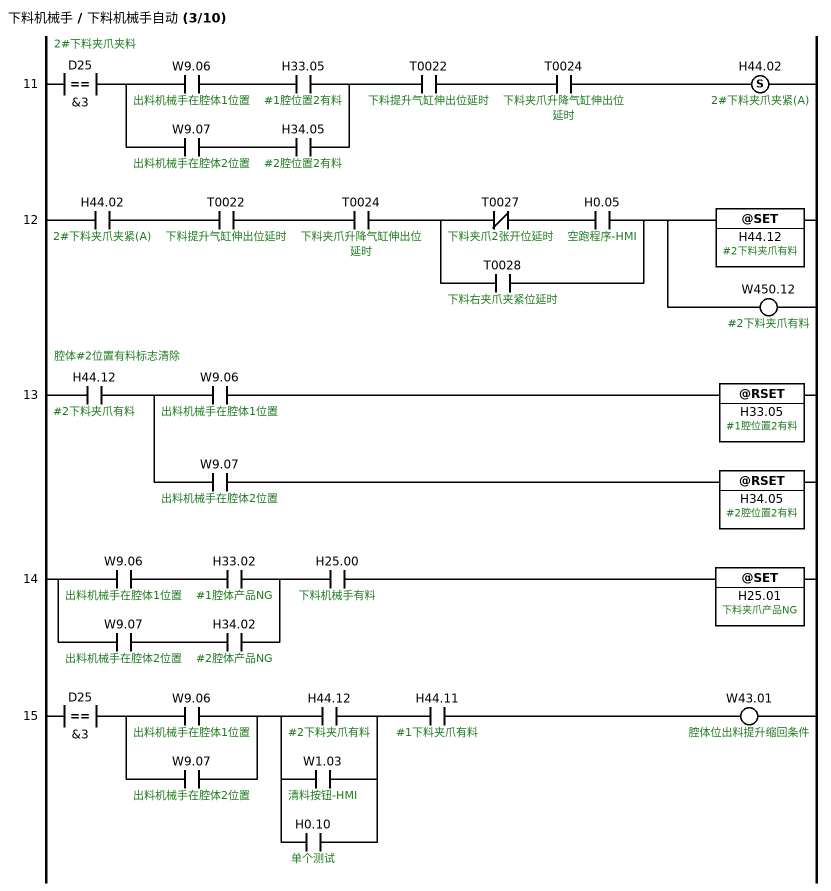
; rung 11: 2#下料夹爪夹料
LD=(300) D25 &3
LD W9.06  ; 出料机械手在腔体1位置
AND H33.05  ; #1腔位置2有料
LD W9.07  ; 出料机械手在腔体2位置
AND H34.05  ; #2腔位置2有料
ORLD
ANDLD
AND T0022  ; 下料提升气缸伸出位延时
AND T0024  ; 下料夹爪升降气缸伸出位延时
SET H44.02  ; 2#下料夹爪夹紧(A)
; rung 12
LD H44.02  ; 2#下料夹爪夹紧(A)
AND T0022  ; 下料提升气缸伸出位延时
AND T0024  ; 下料夹爪升降气缸伸出位延时
LDNOT T0027  ; 下料夹爪2张开位延时
AND H0.05  ; 空跑程序-HMI
OR T0028  ; 下料右夹爪夹紧位延时
ANDLD
@SET H44.12  ; #2下料夹爪有料
OUT W450.12  ; #2下料夹爪有料
; rung 13: 腔体#2位置有料标志清除
LD H44.12  ; #2下料夹爪有料
OUT TR0
AND W9.06  ; 出料机械手在腔体1位置
@RSET H33.05  ; #1腔位置2有料
LD TR0
AND W9.07  ; 出料机械手在腔体2位置
@RSET H34.05  ; #2腔位置2有料
; rung 14
LD W9.06  ; 出料机械手在腔体1位置
AND H33.02  ; #1腔体产品NG
LD W9.07  ; 出料机械手在腔体2位置
AND H34.02  ; #2腔体产品NG
ORLD
AND H25.00  ; 下料机械手有料
@SET H25.01  ; 下料夹爪产品NG
; rung 15
LD=(300) D25 &3
LD W9.06  ; 出料机械手在腔体1位置
OR W9.07  ; 出料机械手在腔体2位置
ANDLD
LD H44.12  ; #2下料夹爪有料
OR W1.03  ; 清料按钮-HMI
OR H0.10  ; 单个测试
ANDLD
AND H44.11  ; #1下料夹爪有料
OUT W43.01  ; 腔体位出料提升缩回条件

